(* IEC 61131-3 sources: Industry-PLC-LLM/data/PLCBEAD_repo/PLCBEAD_PLCEmbed-main/PLC-BEAD/Source/OpenPLCv2 (part 2) *)

(* ---- BAR_GRAPH.ST ---- *)
FUNCTION_BLOCK BAR_GRAPH
	VAR_INPUT
		X :	REAL;
		RST :	BOOL;
		TRIGGER_LOW :	REAL;
		TRIGGER_HIGH :	REAL;
		ALARM_LOW :	BOOL;
		ALARM_HIGH :	BOOL;
		LOG_SCALE :	BOOL;
	END_VAR

	VAR_OUTPUT
		LOW :	BOOL;
		Q1 :	BOOL;
		Q2 :	BOOL;
		Q3 :	BOOL;
		Q4 :	BOOL;
		Q5 :	BOOL;
		Q6 :	BOOL;
		HIGH :	BOOL;
		ALARM :	BOOL;
		STATUS :	BYTE;
	END_VAR

	VAR
		init :	BOOL;
		T1 :	REAL;
		T2 :	REAL;
		T3 :	REAL;
		T4 :	REAL;
		T5 :	REAL;
		temp :	REAL;
	END_VAR

	IF NOT init THEN
		init := TRUE;
		IF log_scale THEN
			temp := EXP(LN(Trigger_high / Trigger_low) * 0.166666666666666666666);
			T1 := trigger_low * temp;
			T2 := T1 * temp;
			T3 := T2 * temp;
			T4 := T3 * temp;
			T5 := T4 * temp;
		ELSE
			temp := (trigger_high - trigger_low) * 0.142857142;
			T1 := trigger_low + temp;
			T2 := T1 + temp;
			T3 := T2 + temp;
			T4 := T3 + temp;
			T5 := T4 + temp;
		END_IF;
	END_IF;

	Q1 := FALSE;
	Q2 := FALSE;
	Q3 := FALSE;
	Q4 := FALSE;
	Q5 := FALSE;
	Q6 := FALSE;
	status := BYTE#110;

	IF NOT alarm_low THEN low := FALSE; END_IF;
	IF NOT alarm_high THEN high := FALSE; END_IF;
	IF rst THEN
		alarm := FALSE;
		low := FALSE;
		high := FALSE;
	END_IF;

	IF X < trigger_low THEN
		Low := TRUE;
		status := BYTE#111;
		IF alarm_low THEN
			alarm := TRUE;
			status := BYTE#1;
		END_IF;
	ELSIF X < T1 THEN
		Q1 := TRUE;
	ELSIF x < t2 THEN
		Q2 := TRUE;
	ELSIF x < t3 THEN
		Q3 := TRUE;
	ELSIF x < T4 THEN
		Q4 := TRUE;
	ELSIF x < T5 THEN
		q5 := TRUE;
	ELSIF x < trigger_high THEN
		q6 := TRUE;
	ELSE
		high := TRUE;
		status := BYTE#112;
		IF alarm_high THEN
			alarm := TRUE;
			status := BYTE#2;
		END_IF;
	END_IF;

END_FUNCTION_BLOCK

PROGRAM program0
  VAR
    LocalVar0 : REAL;
    LocalVar1 : BOOL;
	LocalVar2 : REAL;
	LocalVar3 : REAL;
	LocalVar4 : BOOL;
	LocalVar5 : BOOL;
	LocalVar6 : BOOL;

	LOW   :	BOOL;
	Q1    :	BOOL;
	Q2    :	BOOL;
	Q3    :	BOOL;
	Q4    :	BOOL;
	Q5    :	BOOL;
	Q6    :	BOOL;
	HIGH  :	BOOL;
	ALARM :	BOOL;
	STATUS:	BYTE;

	func_block : BAR_GRAPH;
  END_VAR
	func_block.X := LocalVar0;
	func_block.RST := LocalVar1;
	func_block.TRIGGER_LOW := LocalVar2;
	func_block.TRIGGER_HIGH := LocalVar3;
	func_block.ALARM_LOW := LocalVar4;
	func_block.ALARM_HIGH := LocalVar5;
	func_block.LOG_SCALE := LocalVar6;

	func_block();
	LOW   := func_block.LOW   ;
	Q1    := func_block.Q1    ;
	Q2    := func_block.Q2    ;
	Q3    := func_block.Q3    ;
	Q4    := func_block.Q4    ;
	Q5    := func_block.Q5    ;
	Q6    := func_block.Q6    ;
	HIGH  := func_block.HIGH  ;
	ALARM := func_block.ALARM ;
	STATUS:= func_block.STATUS;

END_PROGRAM

CONFIGURATION Config0
  RESOURCE Res0 ON PLC
    TASK task0(INTERVAL := T#20ms,PRIORITY := 0);
    PROGRAM instance0 WITH task0 : program0;
  END_RESOURCE
END_CONFIGURATION

(* ---- BASE64_DECODE_STREAM.ST ---- *)
TYPE
  oscat_aB0_47	: ARRAY [0..47]	OF BYTE;
  oscat_aB0_63	: ARRAY [0..63]	OF BYTE;
END_TYPE

FUNCTION_BLOCK BASE64_DECODE_STREAM
	VAR_IN_OUT
		BUF1 :	oscat_aB0_63;
		BUF2 :	oscat_aB0_47;
	END_VAR

	VAR_INPUT
		SIZE1 :	INT;
	END_VAR

	VAR_OUTPUT
		SIZE2 :	INT;
	END_VAR

	VAR
		a :	INT;
		b :	WORD;
		o :	INT;
		off :	INT;
		i1 :	INT;
		i2 :	INT;
		c :	INT;
	END_VAR

	IF SIZE1 <= 0 THEN SIZE2 := 0; RETURN; END_IF;
	c := SIZE1 - 1;
	i2 := 0;
	a := 0;
	b := WORD#0;
	FOR i1 := 0 TO c DO
		o := BYTE_TO_INT(BUF1[i1]);
		IF o = 61  (* = *) THEN EXIT;
		ELSIF o > 96 (* a-z *) THEN off := 71;
		ELSIF o > 64 (* A-Z *) THEN off := 65;
		ELSIF o > 47 (* 0-9 *) THEN off := -4;
		ELSIF o = 43 (* + *) THEN off := -19;
		ELSIF o = 47 (* / *) THEN off := -16;
		END_IF;
		b := SHL(b,6) OR INT_TO_WORD(o - off);
		a := a + 6;
		IF a >= 8 THEN
			a := a - 8;
			BUF2[i2] := WORD_TO_BYTE(SHR(b,a));
			i2 := i2 + 1;
			b := b AND NOT SHL(WORD#16#FFFF,a);
		END_IF;
	END_FOR;
	SIZE2 := i2;
END_FUNCTION_BLOCK

PROGRAM program0
  VAR
	BUF1  :	oscat_aB0_63;
	BUF2  :	oscat_aB0_47;

	SIZE1 :	INT;

	SIZE2 :	INT;
	func_block : BASE64_DECODE_STREAM;
  END_VAR
	func_block.BUF1 :=BUF1 ;
	func_block.BUF2 :=BUF2 ;
	func_block.SIZE1:=SIZE1;
	func_block();
	BUF1 := func_block.BUF1;
	BUF2 := func_block.BUF2;
	SIZE2 := func_block.SIZE2;
END_PROGRAM

CONFIGURATION Config0
  RESOURCE Res0 ON PLC
    TASK task0(INTERVAL := T#20ms,PRIORITY := 0);
    PROGRAM instance0 WITH task0 : program0;
  END_RESOURCE
END_CONFIGURATION

(* ---- BLIND_ACTUATOR.ST ---- *)
FUNCTION_BLOCK INTERLOCK_Block

	VAR_INPUT
		I1 :	BOOL;
		I2 :	BOOL;
		TL :	TIME;
	END_VAR

	VAR_OUTPUT
		Q1 :	BOOL;
		Q2 :	BOOL;
	END_VAR

	VAR
		T1 :	TOF;
		T2 :	TOF;
	END_VAR

	T1(IN := I1, PT := TL);
	T2(IN := I2, PT := TL);

	Q1 := I1 AND NOT t2.Q;
	Q2 := I2 AND NOT t1.Q;

END_FUNCTION_BLOCK

FUNCTION TIME_TO_UDINT2:UDINT
	VAR_INPUT
		X :	TIME;
	END_VAR

	TIME_TO_UDINT2 := DINT_TO_UDINT(TIME_TO_DINT(X));
END_FUNCTION

FUNCTION_BLOCK T_PLC_MS_block
	VAR_OUTPUT
		T_PLC_MS :	UDINT;
	END_VAR

	VAR_EXTERNAL
		PLC_TICKS_PER_SEC :	INT;
		PLC_SYS_TICK_CNT :	DINT;
	END_VAR

	VAR
		debug :	BOOL;(*Debug-Mode ON / OFF*)
		N :	INT;(*Debug-Faktor*)
		Offset :	UDINT;(*Debug-Offset*)
		temp :	DWORD := DWORD#1;(*Debug-Offset*)
		mode :	BOOL;(*modus*)
		faktor :	UDINT;(*Systemtakt-Faktor*)
		init :	BOOL;
		v_plc_ticks_per_sec :	UDINT;
		base :	UDINT := UDINT#1000;
	END_VAR

	IF init = FALSE THEN
		v_plc_ticks_per_sec := INT_TO_UDINT(PLC_TICKS_PER_SEC);
		IF v_plc_ticks_per_sec = UDINT#1024 THEN
			faktor := UDINT#1;
			mode := FALSE;
		ELSIF v_plc_ticks_per_sec > UDINT#0 THEN
			IF v_plc_ticks_per_sec <= base THEN
				faktor := base / v_plc_ticks_per_sec;
				mode := FALSE;
			ELSE
				faktor := v_plc_ticks_per_sec / base;
				mode := TRUE;
			END_IF;
		ELSE
			faktor := UDINT#1;
		END_IF;
		init := TRUE;
	END_IF;

	IF mode THEN
		T_PLC_MS := DINT_TO_UDINT(PLC_SYS_TICK_CNT) / faktor;
	ELSE
		T_PLC_MS := DINT_TO_UDINT(PLC_SYS_TICK_CNT) * faktor;
	END_IF;

	IF debug THEN
		T_PLC_MS := (DWORD_TO_UDINT(SHL(UDINT_TO_DWORD(T_PLC_MS),N) OR SHL(temp,N)) - UDINT#1) + Offset;
	END_IF;
END_FUNCTION_BLOCK

FUNCTION FRMP_B:BYTE
	VAR_INPUT
		START :	BYTE;
		DIR :	BOOL;
		TD :	TIME;
		TR :	TIME;
	END_VAR

	IF TD < TR THEN
		FRMP_B := MIN(UDINT_TO_BYTE(DWORD_TO_UDINT(SHL(TIME_TO_DWORD(TD), 8)) / TIME_TO_UDINT2(TR)), SEL(DIR, START, USINT_TO_BYTE(USINT#255 - BYTE_TO_USINT(START))));
		IF DIR THEN
			FRMP_B := USINT_TO_BYTE(BYTE_TO_USINT(START) + BYTE_TO_USINT(FRMP_B));
		ELSE
			FRMP_B := USINT_TO_BYTE(BYTE_TO_USINT(START) - BYTE_TO_USINT(FRMP_B));
		END_IF;
	ELSE
		FRMP_B := SEL(DIR, BYTE#0, BYTE#255);
	END_IF;
END_FUNCTION

FUNCTION_BLOCK _RMP_B
	VAR_INPUT
		DIR :	BOOL;
		E :	BOOL := TRUE;
		TR :	TIME;
	END_VAR

	VAR_IN_OUT
		RMP :	BYTE;
	END_VAR

	VAR
		T_PLC_MS :	T_PLC_MS_block;
		tx :	TIME;
		tl :	TIME;
		tn :	TIME;
		init :	BOOL;
		last_dir :	BOOL;
		start :	BYTE;
	END_VAR

	T_PLC_MS();
	tx := UDINT_TO_TIME(T_PLC_MS.T_PLC_MS);

	IF E AND init AND (dir = last_dir) AND (RMP <> SEL(DIR, BYTE#0, BYTE#255)) AND TR = tn THEN
		RMP := FRMP_B(start, DIR, tx - tl, TR);
	ELSE
		init := TRUE;
		tl := tx;
		tn := tr;
		start := RMP;
	END_IF;
	last_dir := dir;
END_FUNCTION_BLOCK

FUNCTION_BLOCK RMP_B_Block

	VAR_INPUT
		SET :	BOOL;
		PT :	TIME;
		E :	BOOL := TRUE;
		UP :	BOOL := TRUE;
		RST :	BOOL;
	END_VAR

	VAR_OUTPUT
		OUT :	BYTE;
		BUSY :	BOOL;
		HIGH :	BOOL;
		LOW :	BOOL;
	END_VAR

	VAR
		rmp :	_RMP_B;
	END_VAR

	rmp(dir := UP, E := E, TR := PT, RMP := out);
	out := rmp.RMP;

	IF RST THEN
		out := BYTE#0;
	ELSIF SET THEN
		out := BYTE#255;
	END_IF;

low := out = BYTE#0;
high := out = BYTE#255;
busy := NOT (low OR high) AND E;

END_FUNCTION_BLOCK

FUNCTION_BLOCK BLIND_ACTUATOR_Block

	VAR_INPUT
		UP :	BOOL;
		DN :	BOOL;
		S_IN :	BYTE;
		T_UD :	TIME := T#10s;
		T_ANGLE :	TIME := T#3s;
		T_LOCKOUT :	TIME := t#100ms;
	END_VAR

	VAR_OUTPUT
		POS :	BYTE;
		ANG :	BYTE;
		QU :	BOOL;
		QD :	BOOL;
		STATUS :	BYTE;
	END_VAR

	VAR
		position :	RMP_B_Block;
		angle :	RMP_B_Block;
		lock :	INTERLOCK_Block;
	END_VAR

	lock(i1 := UP, I2 := DN, TL := T_lockout);

	angle(e := lock.Q1 OR lock.Q2, UP := lock.Q1, PT := T_Angle);
	position(e := lock.Q1 AND angle.high OR lock.Q2 AND angle.low, up := lock.Q1, PT := T_UD);

	pos := position.Out;
	ang := angle.Out;

	QU := lock.Q1;
	QD := lock.Q2;

	IF UP AND DN THEN
		status := BYTE#1;
	ELSIF UP THEN
		status := BYTE#121;
	ELSIF DN THEN
		status := BYTE#122;
	ELSE
		status := S_IN;
	END_IF;

END_FUNCTION_BLOCK

PROGRAM program0
	VAR
		UP :	BOOL;
		DN :	BOOL;
		S_IN :	BYTE;
		T_UD :	TIME := T#10s;
		T_ANGLE :	TIME := T#3s;
		T_LOCKOUT :	TIME := t#100ms;
		POS :	BYTE;
		ANG :	BYTE;
		QU :	BOOL;
		QD :	BOOL;
		func_block : BLIND_ACTUATOR_Block;
	END_VAR
	func_block.UP := UP;
	func_block.DN := DN;
	func_block.S_IN := S_IN ;
	func_block.T_UD := T_UD;
	func_block.T_ANGLE := T_ANGLE;
	func_block.T_LOCKOUT := T_LOCKOUT;
	func_block();
	POS  := func_block.POS;
	ANG  := func_block.ANG;
	QU  := func_block.QU;
	QD  := func_block.QD;
END_PROGRAM

CONFIGURATION Config0
	VAR_GLOBAL
		PLC_TICKS_PER_SEC :	INT;
		PLC_SYS_TICK_CNT :	DINT;
	END_VAR
  	RESOURCE Res0 ON PLC
    	TASK task0(INTERVAL := T#20ms,PRIORITY := 0);
    	PROGRAM instance0 WITH task0 : program0;
  	END_RESOURCE
END_CONFIGURATION

(* ---- BLIND_CONTROL.ST ---- *)
FUNCTION_BLOCK INTERLOCK_Block

	VAR_INPUT
		I1 :	BOOL;
		I2 :	BOOL;
		TL :	TIME;
	END_VAR

	VAR_OUTPUT
		Q1 :	BOOL;
		Q2 :	BOOL;
	END_VAR

	VAR
		T1 :	TOF;
		T2 :	TOF;
	END_VAR

	T1(IN := I1, PT := TL);
	T2(IN := I2, PT := TL);

	Q1 := I1 AND NOT t2.Q;
	Q2 := I2 AND NOT t1.Q;

END_FUNCTION_BLOCK

FUNCTION TIME_TO_UDINT2:UDINT
	VAR_INPUT
		X :	TIME;
	END_VAR

	TIME_TO_UDINT2 := DINT_TO_UDINT(TIME_TO_DINT(X));
END_FUNCTION

FUNCTION_BLOCK T_PLC_MS_block
	VAR_OUTPUT
		T_PLC_MS :	UDINT;
	END_VAR

	VAR_EXTERNAL
		PLC_TICKS_PER_SEC :	INT;
		PLC_SYS_TICK_CNT :	DINT;
	END_VAR

	VAR
		debug :	BOOL;(*Debug-Mode ON / OFF*)
		N :	INT;(*Debug-Faktor*)
		Offset :	UDINT;(*Debug-Offset*)
		temp :	DWORD := DWORD#1;(*Debug-Offset*)
		mode :	BOOL;(*modus*)
		faktor :	UDINT;(*Systemtakt-Faktor*)
		init :	BOOL;
		v_plc_ticks_per_sec :	UDINT;
		base :	UDINT := UDINT#1000;
	END_VAR

	IF init = FALSE THEN
		v_plc_ticks_per_sec := INT_TO_UDINT(PLC_TICKS_PER_SEC);
		IF v_plc_ticks_per_sec = UDINT#1024 THEN
			faktor := UDINT#1;
			mode := FALSE;
		ELSIF v_plc_ticks_per_sec > UDINT#0 THEN
			IF v_plc_ticks_per_sec <= base THEN
				faktor := base / v_plc_ticks_per_sec;
				mode := FALSE;
			ELSE
				faktor := v_plc_ticks_per_sec / base;
				mode := TRUE;
			END_IF;
		ELSE
			faktor := UDINT#1;
		END_IF;
		init := TRUE;
	END_IF;

	IF mode THEN
		T_PLC_MS := DINT_TO_UDINT(PLC_SYS_TICK_CNT) / faktor;
	ELSE
		T_PLC_MS := DINT_TO_UDINT(PLC_SYS_TICK_CNT) * faktor;
	END_IF;

	IF debug THEN
		T_PLC_MS := (DWORD_TO_UDINT(SHL(UDINT_TO_DWORD(T_PLC_MS),N) OR SHL(temp,N)) - UDINT#1) + Offset;
	END_IF;
END_FUNCTION_BLOCK

FUNCTION FRMP_B:BYTE
	VAR_INPUT
		START :	BYTE;
		DIR :	BOOL;
		TD :	TIME;
		TR :	TIME;
	END_VAR

	IF TD < TR THEN
		FRMP_B := MIN(UDINT_TO_BYTE(DWORD_TO_UDINT(SHL(TIME_TO_DWORD(TD), 8)) / TIME_TO_UDINT2(TR)), SEL(DIR, START, USINT_TO_BYTE(USINT#255 - BYTE_TO_USINT(START))));
		IF DIR THEN
			FRMP_B := USINT_TO_BYTE(BYTE_TO_USINT(START) + BYTE_TO_USINT(FRMP_B));
		ELSE
			FRMP_B := USINT_TO_BYTE(BYTE_TO_USINT(START) - BYTE_TO_USINT(FRMP_B));
		END_IF;
	ELSE
		FRMP_B := SEL(DIR, BYTE#0, BYTE#255);
	END_IF;
END_FUNCTION

FUNCTION_BLOCK _RMP_B
	VAR_INPUT
		DIR :	BOOL;
		E :	BOOL := TRUE;
		TR :	TIME;
	END_VAR

	VAR_IN_OUT
		RMP :	BYTE;
	END_VAR

	VAR
		T_PLC_MS :	T_PLC_MS_block;
		tx :	TIME;
		tl :	TIME;
		tn :	TIME;
		init :	BOOL;
		last_dir :	BOOL;
		start :	BYTE;
	END_VAR

	T_PLC_MS();
	tx := UDINT_TO_TIME(T_PLC_MS.T_PLC_MS);

	IF E AND init AND (dir = last_dir) AND (RMP <> SEL(DIR, BYTE#0, BYTE#255)) AND TR = tn THEN
		RMP := FRMP_B(start, DIR, tx - tl, TR);
	ELSE
		init := TRUE;
		tl := tx;
		tn := tr;
		start := RMP;
	END_IF;
	last_dir := dir;
END_FUNCTION_BLOCK

FUNCTION_BLOCK RMP_B_Block

	VAR_INPUT
		SET :	BOOL;
		PT :	TIME;
		E :	BOOL := TRUE;
		UP :	BOOL := TRUE;
		RST :	BOOL;
	END_VAR

	VAR_OUTPUT
		OUT :	BYTE;
		BUSY :	BOOL;
		HIGH :	BOOL;
		LOW :	BOOL;
	END_VAR

	VAR
		rmp :	_RMP_B;
	END_VAR

	rmp(dir := UP, E := E, TR := PT, RMP := out);
	out := rmp.RMP;

	IF RST THEN
		out := BYTE#0;
	ELSIF SET THEN
		out := BYTE#255;
	END_IF;

low := out = BYTE#0;
high := out = BYTE#255;
busy := NOT (low OR high) AND E;

END_FUNCTION_BLOCK

FUNCTION_BLOCK BLIND_ACTUATOR_Block

	VAR_INPUT
		UP :	BOOL;
		DN :	BOOL;
		S_IN :	BYTE;
		T_UD :	TIME := T#10s;
		T_ANGLE :	TIME := T#3s;
		T_LOCKOUT :	TIME := t#100ms;
	END_VAR

	VAR_OUTPUT
		POS :	BYTE;
		ANG :	BYTE;
		QU :	BOOL;
		QD :	BOOL;
		STATUS :	BYTE;
	END_VAR

	VAR
		position :	RMP_B_Block;
		angle :	RMP_B_Block;
		lock :	INTERLOCK_Block;
	END_VAR

	lock(i1 := UP, I2 := DN, TL := T_lockout);

	angle(e := lock.Q1 OR lock.Q2, UP := lock.Q1, PT := T_Angle);
	position(e := lock.Q1 AND angle.high OR lock.Q2 AND angle.low, up := lock.Q1, PT := T_UD);

	pos := position.Out;
	ang := angle.Out;

	QU := lock.Q1;
	QD := lock.Q2;

	IF UP AND DN THEN
		status := BYTE#1;
	ELSIF UP THEN
		status := BYTE#121;
	ELSIF DN THEN
		status := BYTE#122;
	ELSE
		status := S_IN;
	END_IF;

END_FUNCTION_BLOCK

FUNCTION _BYTE_TO_INT:INT
	VAR_INPUT
		IN :	BYTE;
	END_VAR

	_BYTE_TO_INT := USINT_TO_INT(BYTE_TO_USINT(IN));
END_FUNCTION

FUNCTION_BLOCK BLIND_CONTROL_Block

	VAR_INPUT
		UP :	BOOL;
		DN :	BOOL;
		S_IN :	BYTE;
		PI :	BYTE;
		AI :	BYTE;
		T_UD :	TIME;
		T_ANGLE :	TIME;
		SENS :	BYTE := 5;
		T_LOCKOUT :	TIME := T#100ms;
	END_VAR

	VAR_OUTPUT
		POS :	BYTE;
		ANG :	BYTE;
		MU :	BOOL;
		MD :	BOOL;
		STATUS :	BYTE;
	END_VAR

	VAR
		act :	BLIND_ACTUATOR_Block;
		delta :	BYTE;
		bTimeTest :	BOOL;
		iPos :	BYTE;
		iAngel :	BYTE;
	END_VAR

	IF bTimeTest THEN
		PI:=iPos;
		AI:=iAngel;
		UP:=TRUE;
		DN:=TRUE;
	END_IF;

	act(T_UD:=T_UD, T_ANGLE:=T_ANGLE, T_lockout := T_Lockout);

	IF UP AND DN THEN
		IF _BYTE_TO_INT(act.pos) < _BYTE_TO_INT(pi) - _BYTE_TO_INT(delta) THEN
			act.UP := TRUE;
			act.DN := FALSE;
			delta := BYTE#0;
			STATUS := BYTE#121;
		ELSIF _BYTE_TO_INT(act.pos) > _BYTE_TO_INT(pi) + _BYTE_TO_INT(delta) THEN
			act.UP := FALSE;
			act.DN := TRUE;
			delta := BYTE#0;
			STATUS := BYTE#122;
		ELSIF _BYTE_TO_INT(act.ang) < _BYTE_TO_INT(ai) - _BYTE_TO_INT(delta) AND T_angle > T#100ms THEN
			act.UP := TRUE;
			act.DN := FALSE;
			delta := SHR(sens,2);
			STATUS := BYTE#123;
		ELSIF _BYTE_TO_INT(act.ang) > _BYTE_TO_INT(ai) + _BYTE_TO_INT(delta) AND T_angle > T#100ms THEN
			act.UP := FALSE;
			act.DN := TRUE;
			delta := SHR(sens,2);
			STATUS := BYTE#124;
		ELSE
			act.UP := FALSE;
			act.DN := FALSE;
			delta := sens;
			STATUS := S_IN;
		END_IF;
	ELSE
		act.UP := UP;
		act.DN := DN;
		STATUS := S_IN;
	END_IF;

	act(T_UD:=T_UD, T_ANGLE:=T_ANGLE, T_lockout := T_Lockout);
	pos := act.pos;
	ang := act.ang;
	MU := act.QU;
	md := act.QD;
	status := act.status;

END_FUNCTION_BLOCK

PROGRAM program0
	VAR
		UP :	BOOL;
		DN :	BOOL;
		S_IN :	BYTE;
		PI :	BYTE;
		AI :	BYTE;
		T_UD :	TIME;
		T_ANGLE :	TIME;
		SENS :	BYTE := 5;
		T_LOCKOUT :	TIME := T#100ms;
		POS :	BYTE;
		ANG :	BYTE;
		MU :	BOOL;
		MD :	BOOL;
		STATUS :	BYTE;
		func_block : BLIND_CONTROL_Block;
	END_VAR
	func_block.UP := UP;
	func_block.DN := DN;
	func_block.S_IN := S_IN ;
	func_block.PI    := PI    ;
	func_block.AI := AI;
	func_block.T_UD := T_UD ;
	func_block.T_ANGLE    := T_ANGLE    ;
	func_block.SENS := SENS;
	func_block.T_LOCKOUT := T_LOCKOUT;
	func_block();
	POS  := func_block.POS;
	ANG  := func_block.ANG;
	MU  := func_block.MU;
	MD  := func_block.MD;
	STATUS  := func_block.STATUS;
END_PROGRAM

CONFIGURATION Config0
	VAR_GLOBAL
		PLC_TICKS_PER_SEC :	INT;
		PLC_SYS_TICK_CNT :	DINT;
	END_VAR
  	RESOURCE Res0 ON PLC
    	TASK task0(INTERVAL := T#20ms,PRIORITY := 0);
    	PROGRAM instance0 WITH task0 : program0;
  	END_RESOURCE
END_CONFIGURATION

(* ---- BLIND_CONTROL_S.ST ---- *)
FUNCTION UDINT_TO_TIME2:TIME

	VAR_INPUT
		IN :	UDINT;
	END_VAR

	UDINT_TO_TIME2 := DINT_TO_TIME(UDINT_TO_DINT(IN));

END_FUNCTION

FUNCTION_BLOCK T_PLC_MS_block
	VAR_OUTPUT
		T_PLC_MS :	UDINT;
	END_VAR

	VAR_EXTERNAL
		PLC_TICKS_PER_SEC :	INT;
		PLC_SYS_TICK_CNT :	DINT;
	END_VAR

	VAR
		debug :	BOOL;(*Debug-Mode ON / OFF*)
		N :	INT;(*Debug-Faktor*)
		Offset :	UDINT;(*Debug-Offset*)
		temp :	DWORD := DWORD#1;(*Debug-Offset*)
		mode :	BOOL;(*modus*)
		faktor :	UDINT;(*Systemtakt-Faktor*)
		init :	BOOL;
		v_plc_ticks_per_sec :	UDINT;
		base :	UDINT := UDINT#1000;
	END_VAR

	IF init = FALSE THEN
		v_plc_ticks_per_sec := INT_TO_UDINT(PLC_TICKS_PER_SEC);
		IF v_plc_ticks_per_sec = UDINT#1024 THEN
			faktor := UDINT#1;
			mode := FALSE;
		ELSIF v_plc_ticks_per_sec > UDINT#0 THEN
			IF v_plc_ticks_per_sec <= base THEN
				faktor := base / v_plc_ticks_per_sec;
				mode := FALSE;
			ELSE
				faktor := v_plc_ticks_per_sec / base;
				mode := TRUE;
			END_IF;
		ELSE
			faktor := UDINT#1;
		END_IF;
		init := TRUE;
	END_IF;

	IF mode THEN
		T_PLC_MS := DINT_TO_UDINT(PLC_SYS_TICK_CNT) / faktor;
	ELSE
		T_PLC_MS := DINT_TO_UDINT(PLC_SYS_TICK_CNT) * faktor;
	END_IF;

	IF debug THEN
		T_PLC_MS := (DWORD_TO_UDINT(SHL(UDINT_TO_DWORD(T_PLC_MS),N) OR SHL(temp,N)) - UDINT#1) + Offset;
	END_IF;
END_FUNCTION_BLOCK

FUNCTION TIME_TO_UDINT2:UDINT
	VAR_INPUT
		X :	TIME;
	END_VAR

	TIME_TO_UDINT2 := DINT_TO_UDINT(TIME_TO_DINT(X));
END_FUNCTION

FUNCTION FRMP_B:BYTE
	VAR_INPUT
		START :	BYTE;
		DIR :	BOOL;
		TD :	TIME;
		TR :	TIME;
	END_VAR

	IF TD < TR THEN
		FRMP_B := MIN(UDINT_TO_BYTE(DWORD_TO_UDINT(SHL(TIME_TO_DWORD(TD), 8)) / TIME_TO_UDINT2(TR)), SEL(DIR, START, USINT_TO_BYTE(USINT#255 - BYTE_TO_USINT(START))));
		IF DIR THEN
			FRMP_B := USINT_TO_BYTE(BYTE_TO_USINT(START) + BYTE_TO_USINT(FRMP_B));
		ELSE
			FRMP_B := USINT_TO_BYTE(BYTE_TO_USINT(START) - BYTE_TO_USINT(FRMP_B));
		END_IF;
	ELSE
		FRMP_B := SEL(DIR, BYTE#0, BYTE#255);
	END_IF;
END_FUNCTION

FUNCTION_BLOCK _RMP_B
	VAR_INPUT
		DIR :	BOOL;
		E :	BOOL := TRUE;
		TR :	TIME;
	END_VAR

	VAR_IN_OUT
		RMP :	BYTE;
	END_VAR

	VAR
		T_PLC_MS :	T_PLC_MS_block;
		tx :	TIME;
		tl :	TIME;
		tn :	TIME;
		init :	BOOL;
		last_dir :	BOOL;
		start :	BYTE;
	END_VAR

	T_PLC_MS();
	tx := UDINT_TO_TIME(T_PLC_MS.T_PLC_MS);

	IF E AND init AND (dir = last_dir) AND (RMP <> SEL(DIR, BYTE#0, BYTE#255)) AND TR = tn THEN
		RMP := FRMP_B(start, DIR, tx - tl, TR);
	ELSE
		init := TRUE;
		tl := tx;
		tn := tr;
		start := RMP;
	END_IF;
	last_dir := dir;
END_FUNCTION_BLOCK

FUNCTION_BLOCK TREND_DW
	VAR_INPUT
		X :	DWORD;
	END_VAR
	VAR_OUTPUT
		Q :	BOOL;
		TU :	BOOL;
		TD :	BOOL;
		D :	DWORD;
	END_VAR

	VAR
		LAST_X :	DWORD;
	END_VAR

	IF X > last_X THEN
		TU := TRUE;
		TD := FALSE;
		D := UDINT_TO_DWORD(DWORD_TO_UDINT(X) - DWORD_TO_UDINT(last_X));
		Q := TRUE;
	ELSIF X < last_X THEN
		TD := TRUE;
		TU := FALSE;
		D := UDINT_TO_DWORD(DWORD_TO_UDINT(last_X) - DWORD_TO_UDINT(X));
		Q := FALSE;
	ELSE
		TU := FALSE;
		TD := FALSE;
		D := DWORD#0;
	END_IF;
	last_X := X;
END_FUNCTION_BLOCK

FUNCTION_BLOCK _RMP_NEXT
	VAR_INPUT
		E :	BOOL := TRUE;
		IN :	BYTE;
		TR :	TIME;
		TF :	TIME;
		TL :	TIME;
	END_VAR

	VAR_OUTPUT
		DIR :	BOOL;
		UP :	BOOL;
		DN :	BOOL;
	END_VAR

	VAR_IN_OUT
		OUT :	BYTE;
	END_VAR
	VAR
		rmx :	_RMP_B;
		dirx :	TREND_DW;
		t_lock :	TP;
		xen :	BOOL;
		xdir :	BOOL;
	END_VAR

	dirx(X := BYTE_TO_DWORD(in));

	t_lock(in := FALSE, pt := TL);

	IF dirx.TU AND (OUT < IN) THEN
		IF NOT xdir AND xen THEN t_lock(in := TRUE); END_IF;
		xen := TRUE;
		xdir := TRUE;
	ELSIF dirx.TD AND (OUT > IN) THEN
		IF xdir AND xen THEN t_lock(in := TRUE); END_IF;
		xen := TRUE;
		xdir := FALSE;
	ELSIF xen THEN
		IF (xdir AND (out >= in)) OR (NOT xdir AND (out <= in)) THEN
			xen := FALSE;
			IF tl > t#0s THEN t_lock(IN := TRUE); END_IF;
		END_IF;
	END_IF;

	IF NOT t_lock.Q AND xen THEN
		UP := XDIR;
		DIR := XDIR;
		DN := NOT XDIR;
	ELSE
		UP := FALSE;
		DN := FALSE;
	END_IF;

	rmx(rmp := OUT, E := E AND (UP OR DN) , dir := DIR, tr := SEL(dir, TF, TR));
	OUT := rmx.RMP;
END_FUNCTION_BLOCK

FUNCTION _BYTE_TO_INT:INT
	VAR_INPUT
		IN :	BYTE;
	END_VAR

	_BYTE_TO_INT := USINT_TO_INT(BYTE_TO_USINT(IN));
END_FUNCTION

FUNCTION_BLOCK BLIND_CONTROL_S_Block

	VAR_INPUT
		UP :	BOOL;
		DN :	BOOL;
		S_IN :	BYTE := BYTE#125;
		PI :	BYTE;
		T_UP :	TIME;
		T_DN :	TIME;
		RU :	BOOL;
		RD :	BOOL;
		T_LOCKOUT :	TIME := T#100ms;
		T_EXT :	TIME;
		EXT_TRIG :	BYTE := BYTE#5;
		R_POS_TOP :	BYTE := BYTE#255;
		R_POS_BOT :	BYTE;
	END_VAR

	VAR_OUTPUT
		POS :	BYTE;
		MU :	BOOL;
		MD :	BOOL;
		STATUS :	BYTE;
	END_VAR

	VAR
		T_PLC_MS :	T_PLC_MS_Block;
		rmp :	_RMP_NEXT;
		tx :	TIME;
		last :	TIME;
		pi_last :	BYTE;
	END_VAR

	T_PLC_MS();
	tx:= UDINT_TO_TIME(T_PLC_MS.T_PLC_MS);

	IF UP  AND NOT DN THEN
		rmp.IN := BYTE#255;
		STATUS := BYTE#121;
	ELSIF DN AND NOT UP THEN
		rmp.IN := BYTE#0;
		STATUS := BYTE#122;
	ELSIF NOT (UP OR DN) THEN
		rmp.IN := PI;
		STATUS := S_IN;
	END_IF;

	rmp(E := UP OR DN, TR := T_UP, TF := T_DN, TL := T_LOCKOUT, OUT := POS);
	pos := rmp.OUT;

	CASE _BYTE_TO_INT(STATUS) OF
		0:
			last := tx;
			PI_last := PI XOR BYTE#255;
			STATUS := BYTE#128;

		121:
			MU := TRUE;
			MD := FALSE;
			IF POS >= USINT_TO_BYTE(USINT#255 - BYTE_TO_USINT(EXT_TRIG)) THEN
				POS := BYTE#255;
				last := tx;
				STATUS := BYTE#129;
			END_IF;

		122:
			MD := TRUE;
			MU := FALSE;
			IF POS <= EXT_TRIG THEN
				POS := BYTE#0;
				last := tx;
				STATUS := BYTE#129;
			END_IF;

		123:
			MD := rmp.DN;
			MU := rmp.UP;
			IF NOT (rmp.DN OR rmp.UP) THEN
				IF POS <= EXT_TRIG THEN
					MD := TRUE;
					last := tx;
					STATUS := BYTE#129;
				ELSIF POS >= USINT_TO_BYTE(USINT#255 - BYTE_TO_USINT(EXT_TRIG)) THEN
					MU := TRUE;
					last := tx;
					STATUS := BYTE#129;
				ELSE
					STATUS := S_IN;
				END_IF;
			END_IF;

		124:
			MD := rmp.DN;
			MU := rmp.UP;
			IF NOT(rmp.DN OR rmp.UP) THEN
				PI_last := PI;
				STATUS := S_IN;
			END_IF;

		127:
			IF (tx - last) >= T_LOCKOUT THEN
					STATUS := S_IN;
			END_IF;

		128:
			MU := TRUE;
			MD := FALSE;
			rmp.IN := BYTE#255;
			IF (tx - last) >= (T_UP +  T_EXT) THEN
				MU := FALSE;
				last := tx;
				STATUS := BYTE#127;
			END_IF;

		129:
			IF (tx - last) >= T_EXT THEN
				MU := FALSE;
				MD := FALSE;
				last := tx;
				STATUS := BYTE#127;
			END_IF;

	ELSE
		MU := FALSE;
		MD := FALSE;
		IF PI <> PI_last THEN
			PI_last := PI;
			rmp.IN := PI;
			STATUS := BYTE#123;
		ELSIF POS = BYTE#0 AND RU THEN
			rmp.IN := R_POS_BOT;
			STATUS := BYTE#124;
		ELSIF pos = BYTE#255 AND RD THEN
			rmp.IN := R_POS_TOP;
			STATUS := BYTE#124;
		ELSE
			STATUS := S_IN;
		END_IF;
	END_CASE;

END_FUNCTION_BLOCK

PROGRAM program0
	VAR
		UP :	BOOL;
		DN :	BOOL;
		S_IN :	BYTE := BYTE#125;
		PI :	BYTE;
		T_UP :	TIME;
		T_DN :	TIME;
		RU :	BOOL;
		RD :	BOOL;
		T_LOCKOUT :	TIME := T#100ms;
		T_EXT :	TIME;
		EXT_TRIG :	BYTE := BYTE#5;
		R_POS_TOP :	BYTE := BYTE#255;
		R_POS_BOT :	BYTE;
		POS :	BYTE;
		MU :	BOOL;
		MD :	BOOL;
		STATUS :	BYTE;
		func_block : BLIND_CONTROL_S_Block;
	END_VAR
	func_block.UP := UP;
	func_block.DN := DN;
	func_block.S_IN := S_IN ;
	func_block.PI    := PI    ;
	func_block.T_UP := T_UP;
	func_block.T_DN := T_DN ;
	func_block.RU    := RU    ;
	func_block.RD := RD;
	func_block.T_LOCKOUT := T_LOCKOUT;
	func_block.T_EXT := T_EXT ;
	func_block.EXT_TRIG    := EXT_TRIG    ;
	func_block.R_POS_TOP := R_POS_TOP;
	func_block.R_POS_BOT := R_POS_BOT ;
	func_block();
	POS  := func_block.POS;
	MU  := func_block.MU;
	MD  := func_block.MD;
	STATUS  := func_block.STATUS;
END_PROGRAM

CONFIGURATION Config0
	VAR_GLOBAL
		PLC_TICKS_PER_SEC :	INT;
		PLC_SYS_TICK_CNT :	DINT;
	END_VAR
  	RESOURCE Res0 ON PLC
    	TASK task0(INTERVAL := T#20ms,PRIORITY := 0);
    	PROGRAM instance0 WITH task0 : program0;
  	END_RESOURCE
END_CONFIGURATION

(* ---- BLIND_INPUT.ST ---- *)
FUNCTION UDINT_TO_TIME2:TIME

	VAR_INPUT
		IN :	UDINT;
	END_VAR

	UDINT_TO_TIME2 := DINT_TO_TIME(UDINT_TO_DINT(IN));

END_FUNCTION

FUNCTION_BLOCK T_PLC_MS_block
	VAR_OUTPUT
		T_PLC_MS :	UDINT;
	END_VAR

	VAR_EXTERNAL
		PLC_TICKS_PER_SEC :	INT;
		PLC_SYS_TICK_CNT :	DINT;
	END_VAR

	VAR
		debug :	BOOL;(*Debug-Mode ON / OFF*)
		N :	INT;(*Debug-Faktor*)
		Offset :	UDINT;(*Debug-Offset*)
		temp :	DWORD := DWORD#1;(*Debug-Offset*)
		mode :	BOOL;(*modus*)
		faktor :	UDINT;(*Systemtakt-Faktor*)
		init :	BOOL;
		v_plc_ticks_per_sec :	UDINT;
		base :	UDINT := UDINT#1000;
	END_VAR

	IF init = FALSE THEN
		v_plc_ticks_per_sec := INT_TO_UDINT(PLC_TICKS_PER_SEC);
		IF v_plc_ticks_per_sec = UDINT#1024 THEN
			faktor := UDINT#1;
			mode := FALSE;
		ELSIF v_plc_ticks_per_sec > UDINT#0 THEN
			IF v_plc_ticks_per_sec <= base THEN
				faktor := base / v_plc_ticks_per_sec;
				mode := FALSE;
			ELSE
				faktor := v_plc_ticks_per_sec / base;
				mode := TRUE;
			END_IF;
		ELSE
			faktor := UDINT#1;
		END_IF;
		init := TRUE;
	END_IF;

	IF mode THEN
		T_PLC_MS := DINT_TO_UDINT(PLC_SYS_TICK_CNT) / faktor;
	ELSE
		T_PLC_MS := DINT_TO_UDINT(PLC_SYS_TICK_CNT) * faktor;
	END_IF;

	IF debug THEN
		T_PLC_MS := (DWORD_TO_UDINT(SHL(UDINT_TO_DWORD(T_PLC_MS),N) OR SHL(temp,N)) - UDINT#1) + Offset;
	END_IF;

END_FUNCTION_BLOCK

FUNCTION_BLOCK CLICK_MODE_Block

	VAR_INPUT
		IN :	BOOL;
		T_LONG :	TIME := T#500ms;
	END_VAR

	VAR_OUTPUT
		SINGLE :	BOOL;
		DOUBLE :	BOOL;
		LONG :	BOOL;
		TP_LONG :	BOOL;
	END_VAR

	VAR
		Timer :	TP;
		cnt :	INT;
		last :	BOOL;
	END_VAR

	timer(in := IN, PT := T_LONG);
	single := FALSE;
	double := FALSE;

	IF timer.Q THEN
		IF NOT in AND last THEN	cnt := cnt + 1; END_IF;
	ELSE
		CASE cnt OF
			1 : single := TRUE;
			2 : double := TRUE;
		END_CASE;
		cnt := 0;
	END_IF;
	last := in;
	TP_LONG := NOT timer.Q AND (NOT LONG) AND IN;
	LONG := NOT timer.Q AND in;

END_FUNCTION_BLOCK

FUNCTION _BYTE_TO_INT:INT
	VAR_INPUT
		IN :	BYTE;
	END_VAR

	_BYTE_TO_INT := USINT_TO_INT(BYTE_TO_USINT(IN));
END_FUNCTION

FUNCTION_BLOCK BLIND_INPUT_Block

	VAR_INPUT
		POS :	BYTE;
		ANG :	BYTE;
		S1 :	BOOL;
		S2 :	BOOL;
		IN :	BOOL;
		PI :	BYTE;
		AI :	BYTE;
		SINGLE_SWITCH :	BOOL;
		CLICK_EN :	BOOL := TRUE;
		CLICK_TIME :	TIME := T#500ms;
		MAX_RUNTIME :	TIME := T#60s;
		MANUAL_TIMEOUT :	TIME := T#1h;
		DEBOUNCE_TIME :	TIME := T#20ms;
		DBL_CLK1 :	BOOL := FALSE;
		DBL_POS1 :	BYTE;
		DBL_ANG1 :	BYTE;
		DBL_CLK2 :	BOOL := FALSE;
		DBL_POS2 :	BYTE := BYTE#255;
		DBL_ANG2 :	BYTE := BYTE#255;
		D1_TOGGLE :	BOOL := TRUE;
		D2_TOGGLE :	BOOL := TRUE;
		MASTER_MODE :	BOOL;
	END_VAR

	VAR_OUTPUT
		QU :	BOOL := TRUE;
		QD :	BOOL := TRUE;
		STATUS :	BYTE;
		PO :	BYTE := BYTE#255;
		AO :	BYTE := BYTE#255;
		D1 :	BOOL;
		D2 :	BOOL;
	END_VAR

	VAR
		s1e :	TOF;
		s2e :	TOF;
		s1d :	CLICK_MODE_Block;
		s2d :	CLICK_MODE_Block;
		dir :	BOOL;
		tx :	TIME;
		last :	TIME;
		T_PLC_MS :	T_PLC_MS_Block;
	END_VAR

	T_PLC_MS();
	tx:= UDINT_TO_TIME(T_PLC_MS.T_PLC_MS);

	s1e(in := S1, pt := DEBOUNCE_TIME);
	s2e(in := S2, pt := DEBOUNCE_TIME);
	s1d(in := (s1e.Q AND NOT SINGLE_SWITCH) OR (s1e.Q AND SINGLE_SWITCH AND dir), t_long := CLICK_TIME);
	s2d(in := (s2e.Q AND NOT SINGLE_SWITCH) OR (s1e.Q AND SINGLE_SWITCH AND NOT dir), t_long := CLICK_TIME);

	IF NOT d1_toggle THEN d1 := FALSE; END_IF;
	IF NOT d2_toggle THEN d2 := FALSE; END_IF;

	IF (s1d.LONG AND s2d.LONG) OR (status = BYTE#139) THEN
	status := BYTE#139;
	IF NOT (s1d.LONG OR s2d.LONG)  THEN status := BYTE#130; END_IF;
	ELSIF s1d.tp_LONG THEN
		status := BYTE#132;
	ELSIF s2d.tp_LONG THEN
		status := BYTE#133;
	ELSIF  s1d.SINGLE THEN
		IF click_en THEN
			IF QU XOR QD THEN
				status := BYTE#131;
			ELSE
				status := BYTE#134;
				last := tx;
				dir := NOT dir;
			END_IF;
		END_IF;
	ELSIF  s2d.SINGLE THEN
		IF click_en THEN
			IF QU XOR QD THEN
				status := BYTE#131;
			ELSE
				status := BYTE#135;
				last := tx;
				dir := NOT dir;
			END_IF;
		END_IF;
	ELSIF in THEN
		status := BYTE#136;
		last := tx;
	ELSIF s1d.DOUBLE THEN
		IF dbl_clk1 THEN
			status := BYTE#137;
			last := tx;
		ELSE
			D1 := NOT D1;
		END_IF;
	ELSIF s2d.DOUBLE THEN
		IF dbl_clk2 THEN
			status := BYTE#138;
			last := tx;
		ELSE
			IF single_switch THEN D1 := NOT D1; ELSE D2 := NOT D2; END_IF;
		END_IF;
	END_IF;

	CASE _BYTE_TO_INT(status) OF
		0:
				status := BYTE#130;

		130:
				IF NOT master_mode THEN
					PO := POS;
					AO := ANG;
				END_IF;
				QU := TRUE;
				QD := TRUE;

		131:
				QU := FALSE;
				QD := FALSE;
				PO := POS;
				AO := ANG;
				IF tx - last >= manual_timeout THEN
					status := BYTE#130;
				END_IF;

		132:
				QU := TRUE;
				QD := FALSE;
				PO := POS; AO := ANG;
				last := tx;
				IF NOT s1d.LONG THEN status := BYTE#131; dir := NOT dir; END_IF;

		133:
				QU := FALSE;
				QD := TRUE;
				PO := POS; AO := ANG;
				last := tx;
				IF NOT s2d.LONG THEN	status := BYTE#131; dir := NOT dir; END_IF;

		134:
				QU := TRUE;
				QD := FALSE;
				PO := POS; AO := ANG;
				IF tx - last >= max_runtime THEN status := BYTE#131; END_IF;

		135:
				QU := FALSE;
				QD := TRUE;
				PO := POS; AO := ANG;
				IF tx - last >= max_runtime THEN status := BYTE#131;	END_IF;

		136:
				QU := TRUE;
				QD := TRUE;
				PO := PI; AO := AI;
				IF tx-last >= max_runtime THEN status := BYTE#130; END_IF;

		137:
				QU := TRUE;
				QD := TRUE;
				PO := DBL_POS1;
				AO := DBL_ANG1;
				IF tx - last >= max_runtime THEN status := BYTE#131; END_IF;

		138:
				QU := TRUE;
				QD := TRUE;
				PO := DBL_POS2;
				AO := DBL_ANG2;
				IF tx - last >= max_runtime THEN status := BYTE#131; END_IF;

		139:
				QU := FALSE;
				QD := FALSE;
				PO := POS;
				AO := ANG;

	END_CASE;

END_FUNCTION_BLOCK

PROGRAM program0
	VAR
		POS :	BYTE;
		ANG :	BYTE;
		S1 :	BOOL;
		S2 :	BOOL;
		IN :	BOOL;
		PI :	BYTE;
		AI :	BYTE;
		SINGLE_SWITCH :	BOOL;
		CLICK_EN :	BOOL := TRUE;
		CLICK_TIME :	TIME := T#500ms;
		MAX_RUNTIME :	TIME := T#60s;
		MANUAL_TIMEOUT :	TIME := T#1h;
		DEBOUNCE_TIME :	TIME := T#20ms;
		DBL_CLK1 :	BOOL := FALSE;
		DBL_POS1 :	BYTE;
		DBL_ANG1 :	BYTE;
		DBL_CLK2 :	BOOL := FALSE;
		DBL_POS2 :	BYTE := BYTE#255;
		DBL_ANG2 :	BYTE := BYTE#255;
		D1_TOGGLE :	BOOL := TRUE;
		D2_TOGGLE :	BOOL := TRUE;
		MASTER_MODE :	BOOL;
		QU :	BOOL := TRUE;
		QD :	BOOL := TRUE;
		STATUS :	BYTE;
		PO :	BYTE := BYTE#255;
		AO :	BYTE := BYTE#255;
		D1 :	BOOL;
		D2 :	BOOL;
		func_block : BLIND_INPUT_Block;
	END_VAR
	func_block.POS := POS;
	func_block.ANG := ANG;
	func_block.S1 := S1 ;
	func_block.S2 := S2;
	func_block.IN := IN;
	func_block.PI := PI;
	func_block.AI := AI;
	func_block.SINGLE_SWITCH := SINGLE_SWITCH;
	func_block.CLICK_EN := CLICK_EN ;
	func_block.CLICK_TIME := CLICK_TIME;
	func_block.MAX_RUNTIME := MAX_RUNTIME;
	func_block.MANUAL_TIMEOUT := MANUAL_TIMEOUT;
	func_block.DEBOUNCE_TIME := DEBOUNCE_TIME;
	func_block.DBL_CLK1 := DBL_CLK1;
	func_block.DBL_POS1 := DBL_POS1 ;
	func_block.DBL_ANG1 := DBL_ANG1;
	func_block.DBL_CLK2 := DBL_CLK2;
	func_block.DBL_POS2 := DBL_POS2;
	func_block.DBL_ANG2 := DBL_ANG2;
	func_block.D1_TOGGLE := D1_TOGGLE ;
	func_block.D2_TOGGLE := D2_TOGGLE;
	func_block.MASTER_MODE := MASTER_MODE;
	func_block();
	QU  := func_block.QU;
	QD  := func_block.QD;
	STATUS  := func_block.STATUS;
	PO  := func_block.PO;
	AO  := func_block.AO;
	D1  := func_block.D1;
	D2  := func_block.D2;
END_PROGRAM

CONFIGURATION Config0
	VAR_GLOBAL
		PLC_TICKS_PER_SEC :	INT;
		PLC_SYS_TICK_CNT :	DINT;
	END_VAR
  	RESOURCE Res0 ON PLC
    	TASK task0(INTERVAL := T#20ms,PRIORITY := 0);
    	PROGRAM instance0 WITH task0 : program0;
  	END_RESOURCE
END_CONFIGURATION

(* ---- BLIND_NIGHT.ST ---- *)
FUNCTION TIME_TO_UDINT2:UDINT
	VAR_INPUT
		X :	TIME;
	END_VAR

	TIME_TO_UDINT2 := DINT_TO_UDINT(TIME_TO_DINT(X));
END_FUNCTION

FUNCTION DT_TO_DATE2:UDINT

	VAR_INPUT
		IN :	UDINT;
	END_VAR

	DT_TO_DATE2 := (IN / UDINT#86400) * UDINT#86400;
END_FUNCTION

FUNCTION DT_TO_TOD2:UDINT
	VAR_INPUT
		IN :	UDINT;
	END_VAR

	DT_TO_TOD2 := (IN MOD UDINT#86400) * UDINT#1000;
END_FUNCTION

FUNCTION_BLOCK BLIND_NIGHT_Block

	VAR_INPUT
		UP :	BOOL;
		DN :	BOOL;
		S_IN :	BYTE;
		PI :	BYTE;
		AI :	BYTE;
		E_NIGHT :	BOOL := TRUE;
		E_DAY :	BOOL := TRUE;
		DTIN :	UDINT;
		SUNRISE :	UDINT;
		SUNSET :	UDINT;
		SUNRISE_OFFSET :	TIME;
		SUNSET_OFFSET :	TIME;
		NIGHT_POSITION :	BYTE;
		NIGHT_ANGLE :	BYTE;
	END_VAR

	VAR_OUTPUT
		QU :	BOOL;
		QD :	BOOL;
		STATUS :	BYTE;
		PO :	BYTE;
		AO :	BYTE;
	END_VAR

	VAR
		night :	BOOL;
		last_night :	UDINT;
		last_day :	UDINT;
	END_VAR

	IF NOT (up AND dn) AND night THEN
		night := FALSE;
	ELSIF (DT_TO_TOD2(dtin) > sunset + TIME_TO_UDINT2(sunset_offset)) AND (last_night < DT_TO_DATE2(dtin)) AND NOT night AND e_night THEN
		night := TRUE;
		last_night := DT_TO_DATE2(dtin);
	ELSIF (DT_TO_TOD2(dtin) > sunrise + TIME_TO_UDINT2(sunrise_offset)) AND (last_day < DT_TO_DATE2(dtin)) AND night AND e_day AND (last_night < DT_TO_DATE2(dtin)) THEN
		night := FALSE;
		last_day := DT_TO_DATE2(dtin);
	END_IF;

	IF UP AND DN AND night THEN
		status := BYTE#141;
		po := night_position;
		ao := night_angle;
	ELSE
		QU := UP;
		QD := DN;
		po := pi;
		ao := ai;
		status := s_in;
	END_IF;

END_FUNCTION_BLOCK

PROGRAM program0
	VAR
		UP :	BOOL;
		DN :	BOOL;
		S_IN :	BYTE;
		PI :	BYTE;
		AI :	BYTE;
		E_NIGHT :	BOOL := TRUE;
		E_DAY :	BOOL := TRUE;
		DTIN :	UDINT;
		SUNRISE :	UDINT;
		SUNSET :	UDINT;
		SUNRISE_OFFSET :	TIME;
		SUNSET_OFFSET :	TIME;
		NIGHT_POSITION :	BYTE;
		NIGHT_ANGLE :	BYTE;
		QU :	BOOL;
		QD :	BOOL;
		STATUS :	BYTE;
		PO :	BYTE;
		AO :	BYTE;

		func_block : BLIND_NIGHT_Block;
	END_VAR
	func_block.UP := UP;
	func_block.DN := DN;
	func_block.S_IN := S_IN ;
	func_block.PI    := PI    ;
	func_block.AI := AI;
	func_block.E_NIGHT := E_NIGHT;
	func_block.E_DAY := E_DAY ;
	func_block.DTIN    := DTIN    ;
	func_block.SUNRISE := SUNRISE;
	func_block.SUNSET := SUNSET;
	func_block.SUNRISE_OFFSET := SUNRISE_OFFSET ;
	func_block.SUNSET_OFFSET    := SUNSET_OFFSET    ;
	func_block.NIGHT_POSITION := NIGHT_POSITION ;
	func_block.NIGHT_ANGLE    := NIGHT_ANGLE    ;

	func_block();
	QU  := func_block.QU;
	QD  := func_block.QD;
	STATUS  := func_block.STATUS;
	PO  := func_block.PO;
	AO  := func_block.AO;
END_PROGRAM

CONFIGURATION Config0
	RESOURCE Res0 ON PLC
		TASK task0(INTERVAL := T#20ms,PRIORITY := 0);
		PROGRAM instance0 WITH task0 : program0;
	END_RESOURCE
END_CONFIGURATION

(* ---- BLIND_SCENE.ST ---- *)
TYPE
	oscat_bsa_X                 : ARRAY [0..2]    OF BYTE;
  	oscat_blind_scene_array     : ARRAY [0..15]   OF oscat_bsa_X := [0, 0, 0, 0, 0, 0, 0, 0, 0, 0, 0, 0, 0, 0, 0, 0];
END_TYPE

FUNCTION _BYTE_TO_INT:INT
	VAR_INPUT
		IN :	BYTE;
	END_VAR

	_BYTE_TO_INT := USINT_TO_INT(BYTE_TO_USINT(IN));
END_FUNCTION

FUNCTION_BLOCK BLIND_SCENE_Block

	VAR_INPUT
		UP :	BOOL;
		DN :	BOOL;
		S_IN :	BYTE;
		PI :	BYTE;
		AI :	BYTE;
		ENABLE :	BOOL;
		SWRITE :	BOOL;
		SCENE :	BYTE;
	END_VAR

	VAR_OUTPUT
		QU :	BOOL;
		QD :	BOOL;
		STATUS :	BYTE;
		PO :	BYTE;
		AO :	BYTE;
	END_VAR

	VAR
		x :	INT;
	END_VAR

	VAR RETAIN
		sx :	oscat_blind_scene_array;
	END_VAR

	x := _BYTE_TO_INT(scene AND BYTE#2#0000_1111);

	IF enable AND (sx[x][2] > BYTE#0) AND UP AND DN THEN
		po := sx[x][0];
		ao := sx[x][1];
		status := INT_TO_BYTE(160 + x);
		QU := TRUE;
		QD := TRUE;
	ELSE
		QU := UP;
		QD := DN;
		status := S_IN;
		po := pi;
		ao := ai;
	END_IF;

	IF swrite THEN
		status := BYTE#176;
		sx[x][0] := pi;
		sx[x][1] := ai;
		IF enable THEN sx[x][2] := BYTE#1; ELSE sx[x][2] := BYTE#0; END_IF;
	END_IF;

END_FUNCTION_BLOCK

PROGRAM program0
	VAR
		UP :	BOOL;
		DN :	BOOL;
		S_IN :	BYTE;
		PI :	BYTE;
		AI :	BYTE;
		ENABLE :	BOOL;
		SWRITE :	BOOL;
		SCENE :	BYTE;
		QU :	BOOL;
		QD :	BOOL;
		STATUS :	BYTE;
		PO :	BYTE;
		AO :	BYTE;

		func_block : BLIND_SCENE_Block;
	END_VAR
	func_block.UP := UP;
	func_block.DN := DN;
	func_block.S_IN := S_IN ;
	func_block.PI    := PI    ;
	func_block.AI := AI;
	func_block.ENABLE := ENABLE;
	func_block.SWRITE := SWRITE ;
	func_block.SCENE := SCENE ;

	func_block();
	QU  := func_block.QU;
	QD  := func_block.QD;
	STATUS  := func_block.STATUS;
	PO  := func_block.PO;
	AO  := func_block.AO;
END_PROGRAM

CONFIGURATION Config0
	RESOURCE Res0 ON PLC
		TASK task0(INTERVAL := T#20ms,PRIORITY := 0);
		PROGRAM instance0 WITH task0 : program0;
	END_RESOURCE
END_CONFIGURATION

(* ---- BLIND_SECURITY.ST ---- *)
FUNCTION_BLOCK BLIND_SECURITY_Block

	VAR_INPUT
		UP :	BOOL;
		DN :	BOOL;
		S_IN :	BYTE;
		PI :	BYTE;
		AI :	BYTE;
		FIRE :	BOOL;
		WIND :	BOOL;
		ALARM :	BOOL;
		DOOR :	BOOL;
		RAIN :	BOOL;
		ALARM_UP :	BOOL := TRUE;
		WIND_UP :	BOOL := TRUE;
		RAIN_UP :	BOOL := TRUE;
	END_VAR

	VAR_OUTPUT
		QU :	BOOL;
		QD :	BOOL;
		STATUS :	BYTE;
		PO :	BYTE;
		AO :	BYTE;
	END_VAR

	IF Fire THEN
		QU := TRUE;
		QD := FALSE;
		status := BYTE#111;
	ELSIF Wind THEN
		QU := Wind_up;
		QD := NOT wind_up;
		status := BYTE#112;
	ELSIF alarm THEN
		QU := Alarm_up;
		QD := NOT Alarm_up;
		status := BYTE#113;
	ELSIF Door THEN
		QU := TRUE;
		QD := FALSE;
		status := BYTE#114;
	ELSIF Rain AND NOT (up XOR dn) THEN
		QU := rain_up;
		QD := NOT rain_up;
		status := BYTE#115;
	ELSE
		QU := UP;
		QD := DN;
		status := S_IN;
		po := pi;
		ao := ai;
	END_IF;

END_FUNCTION_BLOCK

PROGRAM program0
	VAR
		UP :	BOOL;
		DN :	BOOL;
		S_IN :	BYTE;
		PI :	BYTE;
		AI :	BYTE;
		FIRE :	BOOL;
		WIND :	BOOL;
		ALARM :	BOOL;
		DOOR :	BOOL;
		RAIN :	BOOL;
		ALARM_UP :	BOOL := TRUE;
		WIND_UP :	BOOL := TRUE;
		RAIN_UP :	BOOL := TRUE;
		QU :	BOOL;
		QD :	BOOL;
		STATUS :	BYTE;
		PO :	BYTE;
		AO :	BYTE;

		func_block : BLIND_SECURITY_Block;
	END_VAR
	func_block.UP := UP;
	func_block.DN := DN;
	func_block.S_IN := S_IN ;
	func_block.PI    := PI    ;
	func_block.AI := AI;
	func_block.FIRE := FIRE;
	func_block.WIND := WIND ;
	func_block.ALARM := ALARM ;
	func_block.DOOR    := DOOR    ;
	func_block.RAIN := RAIN;
	func_block.ALARM_UP := ALARM_UP;
	func_block.WIND_UP := WIND_UP ;
	func_block.RAIN_UP := RAIN_UP ;

	func_block();
	QU  := func_block.QU;
	QD  := func_block.QD;
	STATUS  := func_block.STATUS;
	PO  := func_block.PO;
	AO  := func_block.AO;
END_PROGRAM

CONFIGURATION Config0
	RESOURCE Res0 ON PLC
		TASK task0(INTERVAL := T#20ms,PRIORITY := 0);
		PROGRAM instance0 WITH task0 : program0;
	END_RESOURCE
END_CONFIGURATION

(* ---- BLIND_SET.ST ---- *)
FUNCTION UDINT_TO_TIME2:TIME

	VAR_INPUT
		IN :	UDINT;
	END_VAR

	UDINT_TO_TIME2 := DINT_TO_TIME(UDINT_TO_DINT(IN));

END_FUNCTION

FUNCTION_BLOCK T_PLC_MS_block
	VAR_OUTPUT
		T_PLC_MS :	UDINT;
	END_VAR

	VAR_EXTERNAL
		PLC_TICKS_PER_SEC :	INT;
		PLC_SYS_TICK_CNT :	DINT;
	END_VAR

	VAR
		debug :	BOOL;(*Debug-Mode ON / OFF*)
		N :	INT;(*Debug-Faktor*)
		Offset :	UDINT;(*Debug-Offset*)
		temp :	DWORD := DWORD#1;(*Debug-Offset*)
		mode :	BOOL;(*modus*)
		faktor :	UDINT;(*Systemtakt-Faktor*)
		init :	BOOL;
		v_plc_ticks_per_sec :	UDINT;
		base :	UDINT := UDINT#1000;
	END_VAR

	IF init = FALSE THEN
		v_plc_ticks_per_sec := INT_TO_UDINT(PLC_TICKS_PER_SEC);
		IF v_plc_ticks_per_sec = UDINT#1024 THEN
			faktor := UDINT#1;
			mode := FALSE;
		ELSIF v_plc_ticks_per_sec > UDINT#0 THEN
			IF v_plc_ticks_per_sec <= base THEN
				faktor := base / v_plc_ticks_per_sec;
				mode := FALSE;
			ELSE
				faktor := v_plc_ticks_per_sec / base;
				mode := TRUE;
			END_IF;
		ELSE
			faktor := UDINT#1;
		END_IF;
		init := TRUE;
	END_IF;

	IF mode THEN
		T_PLC_MS := DINT_TO_UDINT(PLC_SYS_TICK_CNT) / faktor;
	ELSE
		T_PLC_MS := DINT_TO_UDINT(PLC_SYS_TICK_CNT) * faktor;
	END_IF;

	IF debug THEN
		T_PLC_MS := (DWORD_TO_UDINT(SHL(UDINT_TO_DWORD(T_PLC_MS),N) OR SHL(temp,N)) - UDINT#1) + Offset;
	END_IF;

END_FUNCTION_BLOCK

FUNCTION_BLOCK BLIND_SET_Block

	VAR_INPUT
		UP :	BOOL;
		DN :	BOOL;
		S_IN :	INT;
		PI :	BYTE;
		AI :	BYTE;
		IN :	BOOL;
		PX :	BYTE;
		AX :	BYTE;
		OVERRIDE_MANUAL :	BOOL;
		RESTORE_POSITION :	BOOL;
		RESTORE_TIME :	TIME := T#60s;
	END_VAR

	VAR_OUTPUT
		QU :	BOOL;
		QD :	BOOL;
		STATUS :	INT;
		PO :	BYTE;
		AO :	BYTE;
	END_VAR

	VAR
		T_PLC_MS :	T_PLC_MS_Block;
		tx :	TIME;
		ps :	BYTE;
		as :	BYTE;
		last :	TIME;
	END_VAR

	T_PLC_MS();
	tx:= UDINT_TO_TIME(T_PLC_MS.T_PLC_MS);

	IF IN THEN
		IF override_manual OR (UP AND DN) THEN
			status := 178;
		END_IF;
	END_IF;

	CASE STATUS OF
		0:
			status := S_IN;

		178:
			PO := PX;
			AO := AX;
			QU := TRUE;
			QD := TRUE;
			IF NOT in THEN
				STATUS := SEL(RESTORE_POSITION, S_IN, 179);
				last := tx;
			END_IF;

		179:
			PO := ps;
			AO := as;
			IF ((PO = PI) AND (AO = AI))  OR tx - last >= RESTORE_TIME THEN
				status := S_IN;
			END_IF;

	ELSE
		PO := PI;
		ps := PI;
		AO := AI;
		as := AI;
		STATUS := S_IN;
		QU := UP;
		QD := DN;
	END_CASE;

END_FUNCTION_BLOCK

PROGRAM program0
	VAR
		UP :	BOOL;
		DN :	BOOL;
		S_IN :	INT;
		PI :	BYTE;
		AI :	BYTE;
		IN :	BOOL;
		PX :	BYTE;
		AX :	BYTE;
		OVERRIDE_MANUAL :	BOOL;
		RESTORE_POSITION :	BOOL;
		RESTORE_TIME :	TIME := T#60s;
		QU :	BOOL;
		QD :	BOOL;
		STATUS :	INT;
		PO :	BYTE;
		AO :	BYTE;

		func_block : BLIND_SET_Block;
	END_VAR
	func_block.UP := UP;
	func_block.DN := DN;
	func_block.S_IN := S_IN ;
	func_block.PI    := PI    ;
	func_block.AI := AI;
	func_block.IN := IN;
	func_block.PX := PX ;
	func_block.AX := AX ;
	func_block.OVERRIDE_MANUAL    := OVERRIDE_MANUAL    ;
	func_block.RESTORE_POSITION := RESTORE_POSITION;
	func_block.RESTORE_TIME := RESTORE_TIME;

	func_block();
	QU  := func_block.QU;
	QD  := func_block.QD;
	STATUS  := func_block.STATUS;
	PO  := func_block.PO;
	AO  := func_block.AO;
END_PROGRAM

CONFIGURATION Config0
	VAR_GLOBAL
		PLC_TICKS_PER_SEC :	INT;
		PLC_SYS_TICK_CNT :	DINT;
	END_VAR
  	RESOURCE Res0 ON PLC
    	TASK task0(INTERVAL := T#20ms,PRIORITY := 0);
    	PROGRAM instance0 WITH task0 : program0;
  	END_RESOURCE
END_CONFIGURATION

(* ---- BLIND_SHADE_S.ST ---- *)
TYPE
  oscat_STRING5               : STRING;
  oscat_STRING30              : STRING;
END_TYPE

TYPE oscat_CALENDAR :
	STRUCT
		UTC : UDINT;				(* world time UTC *)
		LDT : UDINT;				(* local time *)
		LDATE : UDINT;				(* local date *)
		LTOD : UDINT;				(* local time of day *)
		YEAR : INT;					(* year of LDATE *)
		MONTH : INT;				(* month of LDATE *)
		DAY : INT;					(* day of LDATE *)
		WEEKDAY : INT;				(* weekday of LDATE *)
		OFFSET : INT;				(* Time Zone Offset for Local time in minutes *)
		DST_EN : BOOL;				(* daylight savings time enable *)
		DST_ON : BOOL;				(* true when daylight savings time os on *)
		NAME : oscat_string5;		(* name of time zone *)
		LANGUAGE : INT;			    (* language number pls see language setup *)
		LONGITUDE : REAL;			(* longitude of current location *)
		LATITUDE : REAL;			(* latitude of current location *)
		SUN_RISE : UDINT;			(* sun_rise for current location *)
		SUN_SET : UDINT;			(* sun_set for current location *)
		SUN_MIDDAY : UDINT;			(* worldtime when sun stands at south position *)
		SUN_HEIGTH : REAL;			(* suns heigth at midday, south position *)
		SUN_HOR : REAL;				(* sun angle horizontal 0 = north in degrees *)
		SUN_VER : REAL;				(* sun angle vertical above horizon in degrees *)
		NIGHT : BOOL;				(* true between sun_set and sun_rise *)
		HOLIDAY : BOOL;				(* true when holiday *)
		HOLY_NAME : oscat_string30;	(* name of holiday *)
		WORK_WEEK : INT;			(* current work week *)
	END_STRUCT;
END_TYPE

FUNCTION DT_TO_TOD2:UDINT
	VAR_INPUT
		IN :	UDINT;
	END_VAR

	DT_TO_TOD2 := (IN MOD UDINT#86400) * UDINT#1000;
END_FUNCTION

FUNCTION TIME_TO_UDINT2:UDINT
	VAR_INPUT
		X :	TIME;
	END_VAR

	TIME_TO_UDINT2 := DINT_TO_UDINT(TIME_TO_DINT(X));
END_FUNCTION

FUNCTION_BLOCK BLIND_SHADE_S_Block

	VAR_INPUT
		UP :	BOOL;
		DN :	BOOL;
		S_IN :	BYTE;
		PI :	BYTE;
		ENABLE :	BOOL;
		SUN :	BOOL;
		HORZ1 :	REAL := 100.0;
		HORZ2 :	REAL := 260.0;
		VERT :	REAL := 90.0;
		ALERT :	BOOL;
		SUNRISE_OFFSET :	TIME := T#1h;
		SUNSET_PRESET :	TIME := T#1h;
		SHADE_DELAY :	TIME := T#60s;
		SHADE_POS :	BYTE;
		QU :	BOOL;
		QD :	BOOL;
		STATUS :	BYTE;
		PO :	BYTE;
	END_VAR

	VAR_IN_OUT
		CX :	oscat_CALENDAR;
	END_VAR

	VAR
		angle :	REAL;
		sun_delay :	TOF;
	END_VAR

	sun_delay(IN := sun, PT := shade_delay);

	IF ALERT THEN
	QU := TRUE;
	QD := FALSE;
	STATUS := BYTE#152;
	ELSIF UP AND DN AND ENABLE AND sun_delay.Q
	AND (CX.SUN_HOR > HORZ1) AND (CX.SUN_HOR < HORZ2)
	AND (CX.SUN_VER < VERT)
	AND (DT_TO_TOD2(CX.UTC) > CX.SUN_RISE + TIME_TO_UDINT2(sunrise_offset)) AND (DT_TO_TOD2(CX.UTC) < CX.SUN_SET - TIME_TO_UDINT2(sunset_preset)) THEN
	QU := UP;
	QD := DN;
	STATUS := BYTE#151;
	PO := MIN(PI, shade_pos);
	ELSE
	QU := UP;
	QD := DN;
	PO := PI;
	STATUS := S_IN;
	END_IF;

END_FUNCTION_BLOCK

PROGRAM program0
	VAR
		UP :	BOOL;
		DN :	BOOL;
		S_IN :	BYTE;
		PI :	BYTE;
		ENABLE :	BOOL;
		SUN :	BOOL;
		HORZ1 :	REAL := 100.0;
		HORZ2 :	REAL := 260.0;
		VERT :	REAL := 90.0;
		ALERT :	BOOL;
		SUNRISE_OFFSET :	TIME := T#1h;
		SUNSET_PRESET :	TIME := T#1h;
		SHADE_DELAY :	TIME := T#60s;
		SHADE_POS :	BYTE;
		QU :	BOOL;
		QD :	BOOL;
		STATUS :	BYTE;
		PO :	BYTE;
		CX :	oscat_CALENDAR;

		func_block : BLIND_SHADE_S_Block;
	END_VAR
	func_block.UP := UP;
	func_block.DN := DN;
	func_block.S_IN := S_IN ;
	func_block.PI    := PI    ;
	func_block.ENABLE := ENABLE;
	func_block.SUN := SUN;
	func_block.HORZ1 := HORZ1 ;
	func_block.HORZ2 := HORZ2 ;
	func_block.VERT    := VERT    ;
	func_block.ALERT := ALERT;
	func_block.SUNRISE_OFFSET := SUNRISE_OFFSET;
	func_block.SUNSET_PRESET := SUNSET_PRESET ;
	func_block.SHADE_DELAY := SHADE_DELAY ;
	func_block.SHADE_POS    := SHADE_POS    ;
	func_block.QU := QU;
	func_block.QD := QD;
	func_block.STATUS := STATUS ;
	func_block.PO := PO ;
	func_block.CX := CX ;

	func_block();
	CX  := func_block.CX;
END_PROGRAM

CONFIGURATION Config0
	RESOURCE Res0 ON PLC
		TASK task0(INTERVAL := T#20ms,PRIORITY := 0);
		PROGRAM instance0 WITH task0 : program0;
	END_RESOURCE
END_CONFIGURATION

(* ---- BOILER.ST ---- *)
FUNCTION_BLOCK BOILER_Block

	VAR_INPUT
		T_UPPER :	REAL;
		T_LOWER :	REAL;
		PRESSURE :	BOOL := TRUE;
		ENABLE :	BOOL := TRUE;
		REQ_1 :	BOOL;
		REQ_2 :	BOOL;
		BOOST :	BOOL;
		T_UPPER_MIN :	REAL := REAL#50.0;
		T_UPPER_MAX :	REAL := REAL#60.0;
		T_LOWER_ENABLE :	BOOL;
		T_LOWER_MAX :	REAL := REAL#60.0;
		T_REQUEST_1 :	REAL := REAL#70.0;
		T_REQUEST_2 :	REAL := REAL#50.0;
		T_REQUEST_HYS :	REAL := REAL#5.0;
		T_PROTECT_HIGH :	REAL := REAL#80.0;
		T_PROTECT_LOW :	REAL := REAL#10.0;
	END_VAR

	VAR_OUTPUT
		HEAT :	BOOL;
		ERROR :	BOOL;
		STATUS :	BYTE;
	END_VAR

	VAR
		edge :	BOOL;
		boost_mode :	BOOL;
		flag_0 :	BOOL;
		flag_1 :	BOOL;
		flag_2 :	BOOL;
	END_VAR

	IF t_upper > t_protect_high THEN
		status := BYTE#1;
		heat := FALSE;
		error := TRUE;
	ELSIF t_upper < t_protect_low THEN
		status := BYTE#2;
		heat := TRUE;
		error := TRUE;
	ELSIF t_lower > T_protect_high AND t_lower_enable THEN
		status := BYTE#3;
		heat := FALSE;
		error := TRUE;
	ELSIF t_lower < t_protect_low AND t_lower_enable THEN
		status := BYTE#4;
		heat := TRUE;
		error := TRUE;
	ELSIF NOT pressure THEN
		status := BYTE#5;
		heat := FALSE;
		error := TRUE;
	ELSIF req_1 OR req_2 OR enable OR boost THEN
		error := FALSE;

		IF boost AND NOT edge AND t_upper < t_upper_max THEN
			status := BYTE#101;
			heat := TRUE;
			boost_mode := TRUE;
		ELSIF enable AND t_upper < T_upper_min THEN
			status := BYTE#102;
			heat := TRUE;
		ELSIF req_1 AND t_upper < T_request_1 THEN
			status := BYTE#103;
			heat := TRUE;
		ELSIF req_2 AND t_upper < t_request_2 THEN
			status := BYTE#104;
			heat := TRUE;
		END_IF;

		IF heat THEN
			IF (enable OR boost_mode) THEN
				flag_0 := TRUE;
				IF T_lower_enable AND T_lower > T_lower_max THEN
					flag_0 := FALSE;
					boost_mode := FALSE;
				ELSIF NOT T_lower_enable AND T_upper > T_upper_max THEN
					flag_0 := FALSE;
					boost_mode := FALSE;
				END_IF;
			ELSE
				flag_0 := FALSE;
			END_IF;
			flag_1 := (req_1 AND T_upper > T_request_1 + T_request_hys) AND req_1;
			flag_2 := (req_2 AND T_upper > T_request_2 + T_request_hys) AND req_2;

			heat := flag_0 OR flag_1 OR flag_2;
			IF heat = FALSE THEN status := BYTE#100; END_IF;
		END_IF;
	ELSE
		status := BYTE#100;
		heat := FALSE;
		error := FALSE;
	END_IF;
	edge := boost;

END_FUNCTION_BLOCK

PROGRAM program0
	VAR
		T_UPPER :	REAL;
		T_LOWER :	REAL;
		PRESSURE :	BOOL := TRUE;
		ENABLE :	BOOL := TRUE;
		REQ_1 :	BOOL;
		REQ_2 :	BOOL;
		BOOST :	BOOL;
		T_UPPER_MIN :	REAL := REAL#50.0;
		T_UPPER_MAX :	REAL := REAL#60.0;
		T_LOWER_ENABLE :	BOOL;
		T_LOWER_MAX :	REAL := REAL#60.0;
		T_REQUEST_1 :	REAL := REAL#70.0;
		T_REQUEST_2 :	REAL := REAL#50.0;
		T_REQUEST_HYS :	REAL := REAL#5.0;
		T_PROTECT_HIGH :	REAL := REAL#80.0;
		T_PROTECT_LOW :	REAL := REAL#10.0;
		HEAT :	BOOL;
		ERROR :	BOOL;
		STATUS :	BYTE;

		func_block : BOILER_Block;
	END_VAR
	func_block.T_UPPER := T_UPPER;
	func_block.T_LOWER := T_LOWER;
	func_block.PRESSURE := PRESSURE ;
	func_block.ENABLE    := ENABLE    ;
	func_block.REQ_1 := REQ_1;
	func_block.REQ_2 := REQ_2;
	func_block.BOOST := BOOST ;
	func_block.T_UPPER_MIN := T_UPPER_MIN ;
	func_block.T_UPPER_MAX    := T_UPPER_MAX    ;
	func_block.T_LOWER_ENABLE := T_LOWER_ENABLE;
	func_block.T_LOWER_MAX := T_LOWER_MAX;
	func_block.T_REQUEST_1 := T_REQUEST_1 ;
	func_block.T_REQUEST_2 := T_REQUEST_2 ;
	func_block.T_REQUEST_HYS    := T_REQUEST_HYS    ;
	func_block.T_PROTECT_HIGH := T_PROTECT_HIGH;
	func_block.T_PROTECT_LOW := T_PROTECT_LOW;

	func_block();
	HEAT  := func_block.HEAT;
	ERROR  := func_block.ERROR;
	STATUS  := func_block.STATUS;
END_PROGRAM

CONFIGURATION Config0
	RESOURCE Res0 ON PLC
		TASK task0(INTERVAL := T#20ms,PRIORITY := 0);
		PROGRAM instance0 WITH task0 : program0;
	END_RESOURCE
END_CONFIGURATION

(* ---- BUFFER_COMP.ST ---- *)
TYPE
	oscat_arb_0_249 			  : ARRAY [0..249] 	OF BYTE;
END_TYPE

FUNCTION_BLOCK BUFFER_COMP_Block
	VAR_IN_OUT
		PT1 :	oscat_arb_0_249;
	END_VAR

	VAR_INPUT
		SIZE1 :	INT;
	END_VAR

	VAR_IN_OUT
		PT2 :	oscat_arb_0_249;
	END_VAR

	VAR_INPUT
		SIZE2 :	INT;
		START :	INT;
	END_VAR

	VAR_OUTPUT
		BUFFER_COMP :	INT;
	END_VAR

	VAR
		i :	INT;
		j :	INT;
		end :	INT;
		j2 :	INT;
	END_VAR

	IF SIZE2 <= SIZE1 AND SIZE1 > 0 AND SIZE2 > 0 AND START >= 0 THEN
		end := SIZE1 - SIZE2;
		FOR i := START TO end DO
			IF PT1[i] = PT2[0] THEN
				(* first character matches, now compare rest of array *)
				j := 1;
				j2 := j + i;
				WHILE j < SIZE2 DO
					IF PT2[j] <> PT1[j2] THEN EXIT; END_IF;
					j := j + 1;
					j2 := j2 + 1;
				END_WHILE;
				(* when J > size2 a match was found return the position i in buffer1 *)
				IF j = SIZE2 THEN
					BUFFER_COMP := i;
					RETURN;
				END_IF;
			END_IF;
		END_FOR;
	END_IF;
	BUFFER_COMP := -1;

END_FUNCTION_BLOCK

PROGRAM program0
  VAR
    LocalVar0 : oscat_arb_0_249;
    LocalVar1 : INT;
	LocalVar2 : oscat_arb_0_249;
	LocalVar3 : INT;
	LocalVar4 : INT;
	LocalOUT  : INT;
	func_block : BUFFER_COMP_Block;
  END_VAR
	func_block.PT1  := LocalVar0;
	func_block.SIZE1 := LocalVar1;
	func_block.PT2  := LocalVar2;
	func_block.SIZE2 := LocalVar3;
	func_block.START := LocalVar4;
	func_block();
	LocalOUT := func_block.BUFFER_COMP;
	LocalVar0 := func_block.PT1;
	LocalVar2 := func_block.PT1;

END_PROGRAM

CONFIGURATION Config0
  RESOURCE Res0 ON PLC
    TASK task0(INTERVAL := T#20ms,PRIORITY := 0);
    PROGRAM instance0 WITH task0 : program0;
  END_RESOURCE
END_CONFIGURATION

(* ---- BUFFER_COMP_NW.ST ---- *)
TYPE
  oscat_NW_BUF_LONG  : ARRAY [0..4095] OF BYTE;
END_TYPE

FUNCTION_BLOCK BUFFER_COMP_NW
	VAR_IN_OUT
		PT1 :	oscat_NW_BUF_LONG;
	END_VAR

	VAR_INPUT
		SIZE1 :	INT;
	END_VAR

	VAR_IN_OUT
		PT2 :	oscat_NW_BUF_LONG;
	END_VAR

	VAR_INPUT
		SIZE2 :	INT;
		START :	INT;
	END_VAR

	VAR_OUTPUT
		BUFFER_COMP :	INT;
	END_VAR

	VAR
		i :	INT;
		j :	INT;
		end :	INT;
		j2 :	INT;
	END_VAR

	IF SIZE2 <= SIZE1 AND SIZE1 > 0 AND SIZE2 > 0 AND START >= 0 THEN
		end := SIZE1 - SIZE2;
		FOR i := START TO end DO
			IF PT1[i] = PT2[0] THEN
				(* first character matches, now compare rest of array *)
				j := 1;
				j2 := j + i;
				WHILE j < SIZE2 DO
					IF PT2[j] <> PT1[j2] THEN EXIT; END_IF;
					j := j + 1;
					j2 := j2 + 1;
				END_WHILE;
				(* when J > size2 a match was found return the position i in buffer1 *)
				IF j = SIZE2 THEN
					BUFFER_COMP := i;
					RETURN;
				END_IF;
			END_IF;
		END_FOR;
	END_IF;
	BUFFER_COMP := -1;

END_FUNCTION_BLOCK

PROGRAM program0
  VAR
	PT1   :	oscat_NW_BUF_LONG;

	SIZE1 :	INT;

	PT2   : 	oscat_NW_BUF_LONG;

	SIZE2 :	INT;
	START :	INT;

	BUFFER_COMP :	INT;

	func_block : BUFFER_COMP_NW;
  END_VAR
	func_block.PT1  :=PT1  ;
	func_block.SIZE1:=SIZE1;
	func_block.PT2  :=PT2  ;
	func_block.SIZE2:=SIZE2;
	func_block.START:=START;
	func_block();
	BUFFER_COMP := func_block.BUFFER_COMP;
	PT1 := func_block.PT1;
	PT2 := func_block.PT2;

END_PROGRAM

CONFIGURATION Config0
  RESOURCE Res0 ON PLC
    TASK task0(INTERVAL := T#20ms,PRIORITY := 0);
    PROGRAM instance0 WITH task0 : program0;
  END_RESOURCE
END_CONFIGURATION

(* ---- BYTE_TO_BITS.ST ---- *)
FUNCTION BIT_OF_DWORD : BOOL
  VAR_INPUT
    IN : DWORD;
    N : INT;
  END_VAR

  BIT_OF_DWORD := (SHR(in,N) AND 16#00000001) > 0;
END_FUNCTION

FUNCTION_BLOCK BYTE_TO_BITS
	VAR_INPUT
		IN :	BYTE;
	END_VAR

	VAR_OUTPUT
		B0 :	BOOL;
		B1 :	BOOL;
		B2 :	BOOL;
		B3 :	BOOL;
		B4 :	BOOL;
		B5 :	BOOL;
		B6 :	BOOL;
		B7 :	BOOL;
	END_VAR

	B0 := BIT_OF_DWORD(BYTE_TO_DWORD(IN),0); (* IN.X0 *)
	B1 := BIT_OF_DWORD(BYTE_TO_DWORD(IN),1); (* IN.X1 *)
	B2 := BIT_OF_DWORD(BYTE_TO_DWORD(IN),2); (* IN.X2 *)
	B3 := BIT_OF_DWORD(BYTE_TO_DWORD(IN),3); (* IN.X3 *)
	B4 := BIT_OF_DWORD(BYTE_TO_DWORD(IN),4); (* IN.X4 *)
	B5 := BIT_OF_DWORD(BYTE_TO_DWORD(IN),5); (* IN.X5 *)
	B6 := BIT_OF_DWORD(BYTE_TO_DWORD(IN),6); (* IN.X6 *)
	B7 := BIT_OF_DWORD(BYTE_TO_DWORD(IN),7); (* IN.X7 *)
END_FUNCTION_BLOCK

PROGRAM program0
  VAR
	LocalVar0  : BYTE;
	B0 :	BOOL;
	B1 :	BOOL;
	B2 :	BOOL;
	B3 :	BOOL;
	B4 :	BOOL;
	B5 :	BOOL;
	B6 :	BOOL;
	B7 :	BOOL;
	func_block: BYTE_TO_BITS;
  END_VAR

	func_block.IN  := LocalVar0;
	func_block();
	B0 := func_block.B0;
	B1 := func_block.B1;
	B2 := func_block.B2;
	B3 := func_block.B3;
	B4 := func_block.B4;
	B5 := func_block.B5;
	B6 := func_block.B6;
	B7 := func_block.B7;

END_PROGRAM

CONFIGURATION Config0
  RESOURCE Res0 ON PLC
    TASK task0(INTERVAL := T#20ms,PRIORITY := 0);
    PROGRAM instance0 WITH task0 : program0;
  END_RESOURCE
END_CONFIGURATION

(* ---- BYTE_TO_STRB.ST ---- *)
FUNCTION_BLOCK BYTE_TO_STRB_Block
	VAR_INPUT
		IN :	BYTE;
	END_VAR

	VAR_OUTPUT
		BYTE_TO_STRB :	STRING;
	END_VAR

	VAR
		i :	INT;
	END_VAR

	BYTE_TO_STRB := '';
	FOR i := 1 TO 8 DO
		IF (in AND BYTE#2#1000_0000) = BYTE#2#1000_0000 THEN
			BYTE_TO_STRB := CONCAT(BYTE_TO_STRB,'1');
		ELSE
			BYTE_TO_STRB := CONCAT(BYTE_TO_STRB,'0');
		END_IF;
		in := SHL(in, 1);
	END_FOR;

END_FUNCTION_BLOCK

PROGRAM program0
  VAR
    LocalVar0 : BYTE;
	LocalOUT  : STRING;
	func_block : BYTE_TO_STRB_Block;
  END_VAR
	func_block.IN  := LocalVar0;
	func_block();
	LocalOUT := func_block.BYTE_TO_STRB;

END_PROGRAM

CONFIGURATION Config0
  RESOURCE Res0 ON PLC
    TASK task0(INTERVAL := T#20ms,PRIORITY := 0);
    PROGRAM instance0 WITH task0 : program0;
  END_RESOURCE
END_CONFIGURATION

(* ---- BYTE_TO_STRH.ST ---- *)
FUNCTION_BLOCK BYTE_TO_STRH_Block
	VAR_INPUT
		IN :	BYTE;
	END_VAR

	VAR_OUTPUT
		BYTE_TO_STRH :	STRING;
	END_VAR

	BYTE_TO_STRH:=BYTE_TO_STRING(IN);

END_FUNCTION_BLOCK

PROGRAM program0
  VAR
    LocalVar0 : BYTE;
	LocalOUT  : STRING;
	func_block : BYTE_TO_STRH_Block;
  END_VAR
	func_block.IN  := LocalVar0;
	func_block();
	LocalOUT := func_block.BYTE_TO_STRH;

END_PROGRAM

CONFIGURATION Config0
  RESOURCE Res0 ON PLC
    TASK task0(INTERVAL := T#20ms,PRIORITY := 0);
    PROGRAM instance0 WITH task0 : program0;
  END_RESOURCE
END_CONFIGURATION

(* ---- CABS.ST ---- *)
TYPE oscat_complex :
  STRUCT
	re : REAL;
	im : REAL;
  END_STRUCT;
END_TYPE

FUNCTION HYPOT:REAL
	VAR_INPUT
		X :	REAL;
		Y :	REAL;
	END_VAR

	HYPOT := SQRT(x*x + y*y);
END_FUNCTION

FUNCTION_BLOCK CABS_Block
	VAR_INPUT
		X :	oscat_complex;
	END_VAR

	VAR_OUTPUT
		CABS :	REAL;
	END_VAR

	CABS := HYPOT(x.re, x.im);

END_FUNCTION_BLOCK

PROGRAM program0
  VAR
    LocalVar0 : oscat_complex;
	LocalOUT  : REAL;
	func_block : CABS_Block;
  END_VAR
	func_block.X  := LocalVar0;
	func_block();
	LocalOUT := func_block.CABS;

END_PROGRAM

CONFIGURATION Config0
  RESOURCE Res0 ON PLC
    TASK task0(INTERVAL := T#20ms,PRIORITY := 0);
    PROGRAM instance0 WITH task0 : program0;
  END_RESOURCE
END_CONFIGURATION

(* ---- CACOS.ST ---- *)
TYPE oscat_complex :
  STRUCT
	re : REAL;
	im : REAL;
  END_STRUCT;
END_TYPE

FUNCTION ATAN2:REAL
	VAR_INPUT
		X :	REAL;
		Y :	REAL;
	END_VAR

	IF X > 0.0 THEN
		ATAN2 := ATAN(Y/X);
	ELSIF X < 0.0 THEN
		IF Y >= 0.0 THEN
			ATAN2 := ATAN(Y/X) + 3.14159265358979323846264338327950288;
		ELSE
			ATAN2 := ATAN(Y/X) - 3.14159265358979323846264338327950288;
		END_IF;
	ELSIF Y > 0.0 THEN
		ATAN2 := 1.5707963267948965580;
	ELSIF Y < 0.0 THEN
		ATAN2 := -1.5707963267948965580;
	ELSE
		ATAN2 := 0.0;
	END_IF;

END_FUNCTION

FUNCTION HYPOT:REAL
	VAR_INPUT
		X :	REAL;
		Y :	REAL;
	END_VAR

	HYPOT := SQRT(x*x + y*y);
END_FUNCTION

FUNCTION_BLOCK CLOG_Block

	VAR_INPUT
		X :	oscat_complex;
	END_VAR

	VAR_OUTPUT
		CLOG :	oscat_complex;
	END_VAR

	CLOG.re := LN(HYPOT(X.re, X.im));
	CLOG.im := ATAN2(X.im, X.re);

END_FUNCTION_BLOCK

FUNCTION SGN : INT
  VAR_INPUT
    x : REAL;
  END_VAR

  IF X > 0.0 THEN
  	sgn := 1;
  ELSIF X < 0.0 THEN
  	sgn := -1;
  ELSE
  	sgn := 0;
  END_IF;
END_FUNCTION

FUNCTION_BLOCK CSQRT_Block
	VAR_INPUT
		X :	oscat_complex;
	END_VAR

	VAR_OUTPUT
		CSQRT :	oscat_complex;
	END_VAR

	VAR
		temp :	REAL;
	END_VAR

	temp := HYPOT(x.re, x.im);
	CSQRT.re :=  SQRT(0.5 * (temp + x.re));
	CSQRT.im :=  INT_TO_REAL(sgn(x.im)) * SQRT(0.5 * (temp - x.re));

END_FUNCTION_BLOCK

FUNCTION_BLOCK CACOSH_Block
	VAR_INPUT
		X :	oscat_complex;
	END_VAR

	VAR_OUTPUT
		CACOSH :	oscat_complex;
	END_VAR

	VAR
		Y :	oscat_complex;
		CLOG :	CLOG_Block;
		CSQRT :	CSQRT_Block;
	END_VAR

	y.re := (X.re - X.im)*(X.re + X.im) - 1.0;
	y.im := 2.0 * X.re * X.im;
	CSQRT(X:=y);
	y    := CSQRT.CSQRT;
	y.re := y.re + x.re;
	y.im := y.im + x.im;
	CLOG(X:=y);
	CACOSH  := CLOG.CLOG;
END_FUNCTION_BLOCK

FUNCTION_BLOCK CACOS_Block
	VAR_INPUT
		X :	oscat_complex;
	END_VAR

	VAR_OUTPUT
		CACOS :	oscat_complex;
	END_VAR

	VAR
		Y :	oscat_complex;
		CACOSH :	CACOSH_Block;
	END_VAR

	CACOSH(X:=x);
	y := CACOSH.CACOSH;
	CACOS.re := y.im;
	CACOS.im := -y.re;
END_FUNCTION_BLOCK

PROGRAM program0
  VAR
    LocalVar0 : oscat_complex;
	LocalOUT  : oscat_complex;
	func_block : CACOS_Block;
  END_VAR
	func_block.X  := LocalVar0;
	func_block();
	LocalOUT := func_block.CACOS;
END_PROGRAM

CONFIGURATION Config0
  RESOURCE Res0 ON PLC
    TASK task0(INTERVAL := T#20ms,PRIORITY := 0);
    PROGRAM instance0 WITH task0 : program0;
  END_RESOURCE
END_CONFIGURATION

(* ---- CACOSH.ST ---- *)
TYPE oscat_complex :
  STRUCT
	re : REAL;
	im : REAL;
  END_STRUCT;
END_TYPE

FUNCTION ATAN2:REAL
	VAR_INPUT
		X :	REAL;
		Y :	REAL;
	END_VAR

	IF X > 0.0 THEN
		ATAN2 := ATAN(Y/X);
	ELSIF X < 0.0 THEN
		IF Y >= 0.0 THEN
			ATAN2 := ATAN(Y/X) + 3.14159265358979323846264338327950288;
		ELSE
			ATAN2 := ATAN(Y/X) - 3.14159265358979323846264338327950288;
		END_IF;
	ELSIF Y > 0.0 THEN
		ATAN2 := 1.5707963267948965580;
	ELSIF Y < 0.0 THEN
		ATAN2 := -1.5707963267948965580;
	ELSE
		ATAN2 := 0.0;
	END_IF;

END_FUNCTION

FUNCTION HYPOT:REAL
	VAR_INPUT
		X :	REAL;
		Y :	REAL;
	END_VAR

	HYPOT := SQRT(x*x + y*y);
END_FUNCTION

FUNCTION_BLOCK CLOG_Block

	VAR_INPUT
		X :	oscat_complex;
	END_VAR

	VAR_OUTPUT
		CLOG :	oscat_complex;
	END_VAR

	CLOG.re := LN(HYPOT(X.re, X.im));
	CLOG.im := ATAN2(X.im, X.re);

END_FUNCTION_BLOCK

FUNCTION SGN : INT
  VAR_INPUT
    x : REAL;
  END_VAR

  IF X > 0.0 THEN
  	sgn := 1;
  ELSIF X < 0.0 THEN
  	sgn := -1;
  ELSE
  	sgn := 0;
  END_IF;
END_FUNCTION

FUNCTION_BLOCK CSQRT_Block
	VAR_INPUT
		X :	oscat_complex;
	END_VAR

	VAR_OUTPUT
		CSQRT :	oscat_complex;
	END_VAR

	VAR
		temp :	REAL;
	END_VAR

	temp := HYPOT(x.re, x.im);
	CSQRT.re :=  SQRT(0.5 * (temp + x.re));
	CSQRT.im :=  INT_TO_REAL(sgn(x.im)) * SQRT(0.5 * (temp - x.re));

END_FUNCTION_BLOCK

FUNCTION_BLOCK CACOSH_Block
	VAR_INPUT
		X :	oscat_complex;
	END_VAR

	VAR_OUTPUT
		CACOSH :	oscat_complex;
	END_VAR

	VAR
		Y :	oscat_complex;
		CLOG :	CLOG_Block;
		CSQRT :	CSQRT_Block;
	END_VAR

	y.re := (X.re - X.im)*(X.re + X.im) - 1.0;
	y.im := 2.0 * X.re * X.im;
	CSQRT(X:=y);
	y    := CSQRT.CSQRT;
	y.re := y.re + x.re;
	y.im := y.im + x.im;
	CLOG(X:=y);
	CACOSH  := CLOG.CLOG;
END_FUNCTION_BLOCK

PROGRAM program0
  VAR
    LocalVar0 : oscat_complex;
	LocalOUT  : oscat_complex;
	func_block : CACOSH_Block;
  END_VAR
	func_block.X  := LocalVar0;
	func_block();
	LocalOUT := func_block.CACOSH;
END_PROGRAM

CONFIGURATION Config0
  RESOURCE Res0 ON PLC
    TASK task0(INTERVAL := T#20ms,PRIORITY := 0);
    PROGRAM instance0 WITH task0 : program0;
  END_RESOURCE
END_CONFIGURATION

(* ---- CADD.ST ---- *)
TYPE oscat_complex :
  STRUCT
	re : REAL;
	im : REAL;
  END_STRUCT;
END_TYPE

FUNCTION_BLOCK CADD_Block

	VAR_INPUT
		X :	oscat_complex;
		Y :	oscat_complex;
	END_VAR

	VAR_OUTPUT
		CADD :	oscat_complex;
	END_VAR

	CADD.re := x.re + y.re;
	CADD.im := x.im + y.im;

END_FUNCTION_BLOCK

PROGRAM program0
  VAR
    LocalVar0 : oscat_complex;
	LocalVar1 : oscat_complex;
	LocalOUT  : oscat_complex;
	func_block : CADD_Block;
  END_VAR
	func_block.X  := LocalVar0;
	func_block.Y  := LocalVar0;
	func_block();
	LocalOUT := func_block.CADD;
END_PROGRAM

CONFIGURATION Config0
  RESOURCE Res0 ON PLC
    TASK task0(INTERVAL := T#20ms,PRIORITY := 0);
    PROGRAM instance0 WITH task0 : program0;
  END_RESOURCE
END_CONFIGURATION

(* ---- CALENDAR_CALC.ST ---- *)
TYPE oscat_CALENDAR :
	STRUCT
		UTC : UDINT;				(* world time UTC *)
		LDT : UDINT;				(* local time *)
		LDATE : UDINT;				(* local date *)
		LTOD : UDINT;				(* local time of day *)
		YEAR : INT;					(* year of LDATE *)
		MONTH : INT;				(* month of LDATE *)
		DAY : INT;					(* day of LDATE *)
		WEEKDAY : INT;				(* weekday of LDATE *)
		OFFSET : INT;				(* Time Zone Offset for Local time in minutes *)
		DST_EN : BOOL;				(* daylight savings time enable *)
		DST_ON : BOOL;				(* true when daylight savings time os on *)
		NAME : STRING;		(* name of time zone *)
		LANGUAGE : INT;			    (* language number pls see language setup *)
		LONGITUDE : REAL;			(* longitude of current location *)
		LATITUDE : REAL;			(* latitude of current location *)
		SUN_RISE : UDINT;			(* sun_rise for current location *)
		SUN_SET : UDINT;			(* sun_set for current location *)
		SUN_MIDDAY : UDINT;			(* worldtime when sun stands at south position *)
		SUN_HEIGTH : REAL;			(* suns heigth at midday, south position *)
		SUN_HOR : REAL;				(* sun angle horizontal 0 = north in degrees *)
		SUN_VER : REAL;				(* sun angle vertical above horizon in degrees *)
		NIGHT : BOOL;				(* true between sun_set and sun_rise *)
		HOLIDAY : BOOL;				(* true when holiday *)
		HOLY_NAME : STRING;	(* name of holiday *)
		WORK_WEEK : INT;			(* current work week *)
	END_STRUCT;
END_TYPE

TYPE oscat_LANGUAGE:
  STRUCT
    DEFAULT 	: INT;
	LMAX    	: INT;
  END_STRUCT;
END_TYPE

TYPE
	oscat_LOCATION_ELEMENTS	: ARRAY [1..5] OF INT;
END_TYPE

TYPE
  oscat_ELEMENT_WEEKDAYS	: ARRAY [1..7] OF STRING;
  oscat_WEEKDAYS			: ARRAY [1..3]  OF oscat_ELEMENT_WEEKDAYS := [0, 0, 0];
END_TYPE

TYPE oscat_LOCATION:
  STRUCT
    DEFAULT 	: INT;
	LMAX    	: INT;
	LANGUAGE	: oscat_LOCATION_ELEMENTS;
  END_STRUCT;
END_TYPE

TYPE oscat_HOLIDAY_DATA :
  STRUCT
	NAME : STRING;
	DAY : SINT;
	MONTH : SINT;
	USE : SINT;
	PAD_BYTE : BYTE;
  END_STRUCT;
END_TYPE

TYPE
  oscat_HOLIDAY_DATA_0_29 	: ARRAY [0..29] OF oscat_HOLIDAY_DATA;
  oscat_HOLIDAY_DATA_0_49 	: ARRAY [0..49] OF oscat_HOLIDAY_DATA;
END_TYPE

FUNCTION _REAL_TO_UDINT:UDINT

	VAR_INPUT
		X :	REAL;
	END_VAR

	IF REAL_TO_UDINT(0.5) = UDINT#1 THEN
		_REAL_TO_UDINT := REAL_TO_UDINT(x);
	ELSIF X > 0.0 THEN
		_REAL_TO_UDINT := REAL_TO_UDINT(x+0.5);
	ELSIF X < 0.0 THEN
		_REAL_TO_UDINT := REAL_TO_UDINT(x-0.5);
	ELSE
		_REAL_TO_UDINT := UDINT#0;
  	END_IF;
END_FUNCTION

FUNCTION HOUR_TO_TIME:TIME

	VAR_INPUT
		IN :	REAL;
	END_VAR

	hour_to_time := UDINT_TO_TIME(_REAL_TO_UDINT(IN * 3600000.0));
END_FUNCTION

FUNCTION TIME_TO_UDINT2:UDINT
	VAR_INPUT
		X :	TIME;
	END_VAR

	TIME_TO_UDINT2 := DINT_TO_UDINT(TIME_TO_DINT(X));
END_FUNCTION

FUNCTION FLOOR2 : DINT
	VAR_INPUT
		x : REAL;
	END_VAR

	FLOOR2 := REAL_TO_DINT(X);
	IF DINT_TO_REAL(FLOOR2) > X THEN
		FLOOR2 := FLOOR2 - DINT#1;
	END_IF;

END_FUNCTION

FUNCTION MODR:REAL

	VAR_INPUT
		IN :	REAL;
		DIVI :	REAL;
	END_VAR

	IF divi = 0.0 THEN
		MODR := 0.0;
	ELSE
		MODR := in - DINT_TO_REAL(FLOOR2(in / divi)) * divi;
	END_IF;

END_FUNCTION

FUNCTION RAD:REAL

	VAR_INPUT
		DEGG :	REAL;
	END_VAR

	RAD := MODR(0.0174532925199433 * DEGG , 6.283185307179586476);

END_FUNCTION

FUNCTION REFRACTION:REAL

	VAR_INPUT
		ELEV :	REAL;
	END_VAR

	VAR
		tmp :	REAL;
	END_VAR

	tmp := LIMIT(-1.9, elev, 80.0);
	REFRACTION := 0.0174532925199433 / TAN(0.0174532925199433 * (tmp + 10.3 / (tmp + 5.11)));

END_FUNCTION

FUNCTION TOD_TO_REAL2:REAL
	VAR_INPUT
		IN :	UDINT;
	END_VAR
	TOD_TO_REAL2 := UDINT_TO_REAL(IN);
END_FUNCTION

FUNCTION DEG:REAL

	VAR_INPUT
		X :	REAL;
	END_VAR

	DEG := MODR(57.29577951308232 * X, 360.0);
END_FUNCTION

FUNCTION DT_TO_TOD2:UDINT
	VAR_INPUT
		IN :	UDINT;
	END_VAR

	DT_TO_TOD2 := (IN MOD UDINT#86400) * UDINT#1000;
END_FUNCTION

FUNCTION_BLOCK SUN_POS

	VAR_INPUT
		LATITUDE :	REAL;
		LONGITUDE :	REAL;
		UTC :	UDINT;
	END_VAR

	VAR_OUTPUT
		B :	REAL;
		HR :	REAL;
	END_VAR

	VAR
		g :	REAL;
		a :	REAL;
		d :	REAL;
		h :	REAL;
		t1 :	REAL;
		n :	REAL;
		e :	REAL;
		c :	REAL;
		tau :	REAL;
		sin_d :	REAL;
		rlat :	REAL;
		sin_lat :	REAL;
		cos_lat :	REAL;
		cos_tau :	REAL;
		cos_d :	REAL;
		MATH_PI :	REAL := 3.14159265358979323846264338327950288;
		MATH_PI2 :	REAL := 6.28318530717958647692528676655900576;
	END_VAR

	n := UDINT_TO_REAL(UTC - UDINT#946728000) * 0.000011574074074074;
	g :=MODR(6.240040768 + 0.01720197 * n, MATH_PI2);
	d := MODR(4.89495042 + 0.017202792 * n, MATH_PI2) + 0.033423055 * SIN(g) + 0.000349066 * SIN(2.0*g);
	e := 0.409087723 - 0.000000006981317008 * n;
	cos_d := COS(d);
	sin_d := SIN(d);
	a := ATAN(COS(e) * sin_d / cos_d);
	IF cos_d < 0.0 THEN a := a + MATH_PI; END_IF;
	c := ASIN(SIN(e) * sin_d);

	(* also here we must be very careful utc is from 1.1.1970 for step7 the formula must change *)
	tau := RAD(MODR(6.697376 + (n - 0.25) * 0.0657098245037645 + TOD_TO_REAL2(DT_TO_TOD2(utc)) * 0.0000002785383333, 24.0) * 15.0 + longitude) - a;
	rlat := RAD(latitude);
	sin_lat := SIN(rlat);
	cos_lat := COS(rlat);
	cos_tau := COS(tau);
	t1 := cos_tau * sin_lat - TAN(c) * cos_lat;
	B := ATAN(SIN(tau) / t1);
	IF t1 < 0.0 THEN B := B + MATH_PI2; ELSE B := B + MATH_PI; END_IF;
	B := DEG(MODR(B, MATH_PI2));
	h := DEG(ASIN(COS(C) * cos_tau * cos_lat +SIN(c) * sin_lat));
	IF h > 180.0 THEN h := h - 360.0; END_IF;
	(* consider refraction *)
	HR := h + REFRACTION(h);
END_FUNCTION_BLOCK

FUNCTION HOUR_TO_TOD:UDINT
	VAR_INPUT
		IN :	REAL;
	END_VAR

	hour_to_tod := _REAL_TO_UDINT(IN * 3600000.00);
END_FUNCTION

FUNCTION DAY_OF_YEAR:INT
	VAR_INPUT
		IDATE :	DATE;
	END_VAR

	DAY_OF_YEAR := UDINT_TO_INT((DATE_TO_UDINT(idate) / UDINT#86400) MOD UDINT#1461);
	IF DAY_OF_YEAR > 729 THEN
		IF DAY_OF_YEAR > 1095 THEN DAY_OF_YEAR := DAY_OF_YEAR - 1095; ELSE DAY_OF_YEAR := DAY_OF_YEAR - 729; END_IF;
	ELSIF DAY_OF_YEAR > 364 THEN
		DAY_OF_YEAR := DAY_OF_YEAR - 364;
	ELSE
		DAY_OF_YEAR := DAY_OF_YEAR + 1;
	END_IF;
END_FUNCTION

FUNCTION DAY_OF_YEAR_UDINT:INT
	VAR_INPUT
		IDATE :	UDINT;
	END_VAR

	DAY_OF_YEAR_UDINT := UDINT_TO_INT((idate / UDINT#86400) MOD UDINT#1461);
	IF DAY_OF_YEAR_UDINT > 729 THEN
		IF DAY_OF_YEAR_UDINT > 1095 THEN DAY_OF_YEAR_UDINT := DAY_OF_YEAR_UDINT - 1095; ELSE DAY_OF_YEAR_UDINT := DAY_OF_YEAR_UDINT - 729; END_IF;
	ELSIF DAY_OF_YEAR_UDINT > 364 THEN
		DAY_OF_YEAR_UDINT := DAY_OF_YEAR_UDINT - 364;
	ELSE
		DAY_OF_YEAR_UDINT := DAY_OF_YEAR_UDINT + 1;
	END_IF;
END_FUNCTION

FUNCTION SUN_MIDDAY:UDINT
	VAR_INPUT
		LON :	REAL;
		UTC :	DATE;
	END_VAR

	VAR
		T :	REAL;
		OFFSET :	REAL;
	END_VAR

	T := INT_TO_REAL(DAY_OF_YEAR(utc));
	OFFSET := -0.1752 * SIN(0.033430 * T + 0.5474) - 0.1340 * SIN(0.018234 * T - 0.1939);
	SUN_MIDDAY := HOUR_TO_TOD(12.0 - OFFSET - lon * 0.0666666666666);
END_FUNCTION

FUNCTION SUN_MIDDAY_UDINT:UDINT
	VAR_INPUT
		LON :	REAL;
		UTC :	UDINT;
	END_VAR

	VAR
		T :	REAL;
		OFFSET :	REAL;
	END_VAR

	T := INT_TO_REAL(DAY_OF_YEAR_UDINT(utc));
	OFFSET := -0.1752 * SIN(0.033430 * T + 0.5474) - 0.1340 * SIN(0.018234 * T - 0.1939);
	SUN_MIDDAY_UDINT := HOUR_TO_TOD(12.0 - OFFSET - lon * 0.0666666666666);
END_FUNCTION

FUNCTION_BLOCK SUN_TIME_Block

	VAR_INPUT
		LATITUDE :	REAL;
		LONGITUDE :	REAL;
		UTC :	UDINT;
		H :	REAL := -0.83333333333;
	END_VAR

	VAR_OUTPUT
		MIDDAY :	UDINT;
		SUN_RISE :	UDINT;
		SUN_SET :	UDINT;
		SUN_DECLINATION :	REAL;
	END_VAR

	VAR
		DK :	REAL;
		delta :	UDINT;
		B :	REAL;
	END_VAR

	B := latitude * 0.0174532925199433;
	MIDDAY := SUN_MIDDAY_UDINT(longitude, utc);
	DK := 0.40954 * SIN(0.0172 * (INT_TO_REAL(DAY_OF_YEAR_UDINT(utc)) - 79.35));
	sun_declination := DEG(DK);
	IF sun_declination > 180.0 THEN sun_declination := sun_declination - 360.0; END_IF;
	sun_declination := 90.0 - LATITUDE + sun_declination;
	delta := TIME_TO_UDINT2(HOUR_TO_TIME(ACOS((SIN(RAD(H)) - SIN(B) * SIN(DK)) / (COS(B) * COS(DK))) * 3.819718632));
	sun_rise := MIDDAY - delta;
	sun_set := MIDDAY + delta;
END_FUNCTION_BLOCK

FUNCTION_BLOCK SETUP_LANGUAGE_Block

	VAR_IN_OUT
		LANGUAGE :	oscat_LANGUAGE;
	END_VAR

	VAR
		init :	BOOL;
	END_VAR

	IF init THEN RETURN; END_IF;
	init := TRUE;

	LANGUAGE.DEFAULT  := 1; (* 1=english, 2=german 3=french *)
	LANGUAGE.LMAX := 3;
END_FUNCTION_BLOCK

FUNCTION_BLOCK SETUP_LOCATION
	VAR_IN_OUT
		LOCATION :	oscat_LOCATION;
	END_VAR

	VAR
		init :	BOOL;
	END_VAR

	IF init THEN RETURN; END_IF;
	init := TRUE;

	LOCATION.DEFAULT  := 1;
	LOCATION.LMAX := 5;

	LOCATION.LANGUAGE[1] := 2;
	LOCATION.LANGUAGE[2] := 2;
	LOCATION.LANGUAGE[3] := 3;
	LOCATION.LANGUAGE[4] := 2;
	LOCATION.LANGUAGE[5] := 2;
END_FUNCTION_BLOCK

FUNCTION_BLOCK SETUP_WEEKDAYS

	VAR_IN_OUT
		WEEKDAYS :	oscat_WEEKDAYS;
	END_VAR

	VAR
		init :	BOOL;
	END_VAR

	IF init THEN RETURN; END_IF;
	init := TRUE;

	WEEKDAYS[1][01] := 'Monday';
	WEEKDAYS[1][02] := 'Tuesday';
	WEEKDAYS[1][03] := 'Wednesday';
	WEEKDAYS[1][04] := 'Thursday';
	WEEKDAYS[1][05] := 'Friday';
	WEEKDAYS[1][06] := 'Saturday';
	WEEKDAYS[1][07] := 'Sunday';

	WEEKDAYS[2][01] := 'Montag';
	WEEKDAYS[2][02] := 'Dienstag';
	WEEKDAYS[2][03] := 'Mittwoch';
	WEEKDAYS[2][04] := 'Donnerstag';
	WEEKDAYS[2][05] := 'Freitag';
	WEEKDAYS[2][06] := 'Samstag';
	WEEKDAYS[2][07] := 'Sonntag';

	WEEKDAYS[3][01] := 'Lundi';
	WEEKDAYS[3][02] := 'Mardi';
	WEEKDAYS[3][03] := 'Mercredi';
	WEEKDAYS[3][04] := 'Jeudi';
	WEEKDAYS[3][05] := 'Vendredi';
	WEEKDAYS[3][06] := 'Samedi';
	WEEKDAYS[3][07] := 'Dimanche';
END_FUNCTION_BLOCK

FUNCTION YEAR_OF_DATE:INT
	VAR_INPUT
		IDATE :	UDINT;
	END_VAR

	YEAR_OF_DATE := UDINT_TO_INT((idate+UDINT#43200) / UDINT#31557600 + UDINT#1970);
END_FUNCTION

FUNCTION _INT_TO_UDINT:UDINT
	VAR_INPUT
		IN :	INT;
	END_VAR

	_INT_TO_UDINT := DINT_TO_UDINT(INT_TO_DINT(IN));
END_FUNCTION

FUNCTION SET_DATE:UDINT

	VAR_INPUT
		YEAR :	INT;
		MONTH :	INT;
		DAY :	INT;
	END_VAR

	VAR
		count :	INT;
	END_VAR

	IF month > 2 THEN
		count := (month - 1) * 30;
		IF month > 7 THEN
			count := count + DWORD_TO_INT(SHR(DINT_TO_DWORD(INT_TO_DINT(month) - INT_TO_DINT(3)),1));
		ELSE
			count := count + DWORD_TO_INT(SHR(DINT_TO_DWORD(INT_TO_DINT(month) - INT_TO_DINT(4)),1));
		END_IF;
		IF SHL(INT_TO_WORD(year),14) = WORD#0 THEN
			count := count + 1;
		END_IF;
	ELSE
		count := (month - 1) * 31;
	END_IF;
	SET_DATE := (_INT_TO_UDINT(count + day - 1) + DWORD_TO_UDINT(SHR(UDINT_TO_DWORD(_INT_TO_UDINT(year) * UDINT#1461 - UDINT#2878169), 2))) * UDINT#86400;
END_FUNCTION

FUNCTION DAY_OF_WEEK:INT
	VAR_INPUT
		IDATE :	UDINT;
	END_VAR

	DAY_OF_WEEK := UDINT_TO_INT((idate / UDINT#86400 + UDINT#3) MOD UDINT#7) + INT#01;
END_FUNCTION

FUNCTION EASTER:UDINT
	VAR_INPUT
		YEAR :	INT;
	END_VAR

	VAR
		b :	INT;
		c :	INT;
		oday :	INT;
	END_VAR

	b := (204 - 11 * (year MOD 19)) MOD 30;
	IF b > 27 THEN b := b - 1; END_IF;
	c := (year + WORD_TO_INT(SHR(INT_TO_WORD(year),2)) + b - 13) MOD 7;
	oday := 28 + b - c;
	IF oday > 33 THEN
		easter := set_Date(year, 4, oday - 31);
	ELSE
		easter := set_Date(year, 3, oday);
	END_IF;
END_FUNCTION

FUNCTION LEAP_OF_DATE:BOOL

	VAR_INPUT
		IDATE :	UDINT;
	END_VAR

	LEAP_OF_DATE := SHL(UDINT_TO_DWORD((idate + UDINT#43200) / UDINT#31557600), 30) = DWORD#16#80000000;
END_FUNCTION

FUNCTION MONTH_OF_DATE:INT

	VAR_INPUT
		IDATE :	UDINT;
	END_VAR

	MONTH_OF_DATE := DAY_OF_YEAR_UDINT(idate);
	IF MONTH_OF_DATE < 32 THEN
		MONTH_OF_DATE := 1;
	ELSIF LEAP_OF_DATE((IDATE)) THEN
		MONTH_OF_DATE := (MONTH_OF_DATE * 53 + 1668) / 1623;
	ELSE
		MONTH_OF_DATE := (MONTH_OF_DATE * 53 + 1700) / 1620;
	END_IF;
END_FUNCTION

FUNCTION DAY_OF_MONTH:INT
	VAR_INPUT
		IDATE :	UDINT;
	END_VAR

	day_of_month := DAY_OF_YEAR_UDINT(idate);

	IF leap_of_Date((idate)) THEN
		CASE day_of_month OF
			32..60	:	day_of_month := day_of_month - 31;
			61..91	:	day_of_month := day_of_month - 60;
			92..121 :	day_of_month := day_of_month - 91;
			122..152:	day_of_month := day_of_month - 121;
			153..182:	day_of_month := day_of_month - 152;
			183..213:	day_of_month := day_of_month - 182;
			214..244:	day_of_month := day_of_month - 213;
			245..274:	day_of_month := day_of_month - 244;
			275..305:	day_of_month := day_of_month - 274;
			306..335:	day_of_month := day_of_month - 305;
			336..366:	day_of_month := day_of_month - 335;
		END_CASE;
	ELSE
		CASE day_of_month OF
			32..59	:	day_of_month := day_of_month - 31;
			60..90	:	day_of_month := day_of_month - 59;
			91..120 :	day_of_month := day_of_month - 90;
			121..151:	day_of_month := day_of_month - 120;
			152..181:	day_of_month := day_of_month - 151;
			182..212:	day_of_month := day_of_month - 181;
			213..243:	day_of_month := day_of_month - 212;
			244..273:	day_of_month := day_of_month - 243;
			274..304:	day_of_month := day_of_month - 273;
			305..334:	day_of_month := day_of_month - 304;
			335..365:	day_of_month := day_of_month - 334;
		END_CASE;
	END_IF;
END_FUNCTION

FUNCTION DATE_ADD:UDINT
	VAR_INPUT
		IDATE :	UDINT;
		D :	INT;
		W :	INT;
		M :	INT;
		Y :	INT;
	END_VAR

	VAR
		mo :	INT;
		yr :	INT;
		dm :	INT;
	END_VAR

	DATE_ADD := IDATE + INT_TO_UDINT(D + W * 7) * UDINT#86400;
	yr := Y + YEAR_OF_DATE(DATE_ADD);
	mo := M + MONTH_OF_DATE(DATE_ADD);
	dm := DAY_OF_MONTH(DATE_ADD);
	WHILE mo > 12 DO
		mo := mo - 12;
		yr := yr + 1;
	END_WHILE;
	WHILE mo < 1 DO
		mo := mo + 12;
		yr := yr - 1;
	END_WHILE;
	DATE_ADD := SET_DATE(yr, mo, dm);
END_FUNCTION

FUNCTION DT_TO_DATE2:UDINT
	VAR_INPUT
		IN :	UDINT;
	END_VAR

	DT_TO_DATE2 := (IN / UDINT#86400) * UDINT#86400;
END_FUNCTION

FUNCTION DAY_OF_DATE:DINT
	VAR_INPUT
		IDATE :	UDINT;
	END_VAR

	day_of_date := UDINT_TO_DINT(idate / UDINT#86400);
END_FUNCTION

FUNCTION LEAP_YEAR:BOOL

  VAR_INPUT
    YEAR :	INT;
  END_VAR

  IF (year MOD INT#400) = INT#00 THEN
    leap_year := TRUE;
  ELSIF (year MOD INT#100) = INT#00 THEN
    leap_year := FALSE;
  ELSIF (year MOD INT#04) = INT#00 THEN
    leap_year := TRUE;
  ELSE
    leap_year := FALSE;
  END_IF;

END_FUNCTION

FUNCTION HOUR:INT
	VAR_INPUT
		ITOD :	UDINT;
	END_VAR
	hour := UDINT_TO_INT(itod / UDINT#3600000);
END_FUNCTION

FUNCTION SET_DT:UDINT

	VAR_INPUT
		YEAR : INT;
		MONTH :	INT;
		DAY : INT;
		HOURR : INT;
		MINUTE : INT;
		SECOND : INT;
	END_VAR

	SET_DT := SET_DATE(YEAR, MONTH, DAY) + _INT_TO_UDINT(SECOND) + _INT_TO_UDINT(MINUTE) * UDINT#60 + _INT_TO_UDINT(HOURR) * UDINT#3600;

END_FUNCTION

FUNCTION DST:BOOL
	VAR_INPUT
		UTC :	UDINT;
	END_VAR

	VAR
		yr :	INT;
		yr4 :	UDINT;
		ltc :	UDINT;
		idate :	UDINT;
	END_VAR

	yr := YEAR_OF_DATE(DT_TO_DATE2(UTC));
	ltc := UTC;
	idate := SET_DT(yr, 3, 31, 1, 0, 0);
	yr4 := DWORD_TO_UDINT(SHR(INT_TO_DWORD(5 * yr), 2)) + UDINT#1;
	DST := (idate - ((yr4 + UDINT#3) MOD UDINT#7) * UDINT#86400 <= ltc) AND (idate + (UDINT#214 - (yr4) MOD UDINT#7) * UDINT#86400 > ltc);

END_FUNCTION

FUNCTION UTC_TO_LTIME:UDINT

	VAR_INPUT
		UTC :	UDINT;
		DST_ENABLE :	BOOL;
		TIME_ZONE_OFFSET :	INT;
	END_VAR

	VAR
		tmp :	INT;
	END_VAR

	UTC_TO_LTIME := UTC + _INT_TO_UDINT(TIME_ZONE_OFFSET) * UDINT#60 + BOOL_TO_UDINT(DST_ENABLE AND DST(UTC)) * UDINT#3600;

	tmp := TIME_ZONE_OFFSET * 60 + BOOL_TO_INT(DST_ENABLE AND DST(UTC)) * 3600;
	IF tmp < 0 THEN
		UTC_TO_LTIME := UTC - _INT_TO_UDINT(ABS(tmp));
	ELSE
		UTC_TO_LTIME := UTC + _INT_TO_UDINT(tmp);
	END_IF;

END_FUNCTION

FUNCTION YEAR_BEGIN:UDINT
	VAR_INPUT
		Y :	INT;
	END_VAR
	year_begin := DWORD_TO_UDINT(SHR(UDINT_TO_DWORD(_INT_TO_UDINT(y) * UDINT#1461 - UDINT#2878169),2))*UDINT#86400;

END_FUNCTION

FUNCTION WORK_WEEK:INT

	VAR_INPUT
		IDATE :	UDINT;
	END_VAR

	VAR
		d1 :	UDINT;
		w1 :	INT;
		ds :	UDINT;
		yr :	INT;
		w31 :	INT;
		w01 :	INT;
		wm :	INT;
	END_VAR

	yr := YEAR_OF_DATE(idate);
	d1 := year_begin(yr);
	w1 := DAY_OF_WEEK(d1);
	IF w1 < 5 THEN
		ds := d1 - _INT_TO_UDINT(w1+6) * UDINT#86400;
	ELSE
		ds := d1 + _INT_TO_UDINT(1-w1) * UDINT#86400;
	END_IF;

	work_week := UDINT_TO_INT((idate - ds) / UDINT#604800);

	IF work_week = 0 THEN
		IF w1 > 1 THEN w31 := w1 - 1; ELSE W31 := 7; END_IF;
		IF leap_year(yr - 1) THEN IF w31 > 1 THEN w01 := W31 - 1; ELSE w1 := 7; END_IF; END_IF;
		WORK_WEEK := 52 + BOOL_TO_INT(w31 = 4 OR w01 = 4);
	ELSE
		IF leap_year(yr) THEN
			IF w1 < 7 THEN w31 := w1 + 1; ELSE w31 := 1; END_IF;
		ELSE
			w31 := w1;
		END_IF;
		wm := 52 + BOOL_TO_INT(w31 = 4 OR w1 = 4);
		IF work_week > wm THEN work_week := 1; END_IF;
	END_IF;

END_FUNCTION

FUNCTION_BLOCK HOLIDAY_Block
	VAR_INPUT
		DATE_IN :	UDINT;
		LANGU :	INT;
		FRIDAY :	BOOL;
		SATURDAY :	BOOL;
		SUNDAY :	BOOL;
	END_VAR

	VAR_IN_OUT
		HOLIDAYS :	oscat_HOLIDAY_DATA_0_29;
	END_VAR

	VAR_OUTPUT
		Y :	BOOL;
		NAME :	STRING;
	END_VAR

	VAR
		size :	INT := INT#29;
		last_active :	UDINT;
		ostern :	UDINT;
		i :	INT;
		jahr :	INT;
		x_date :	UDINT;
		lx :	INT;
		wdx :	INT;
		SETUP_LOCATIONS :	SETUP_LOCATION;
		SETUP_WEEKDAYSS :	SETUP_WEEKDAYS;
		SETUP_LANGUAGES :	SETUP_LANGUAGE_Block;
		LOCATION :	oscat_LOCATION;
		WEEKDAYS :	oscat_WEEKDAYS;
		LANGUAGE :	oscat_LANGUAGE;
		wd :	INT;
	END_VAR

	IF last_active = date_in THEN RETURN; END_IF;
	last_active := DATE_IN;

	SETUP_LOCATIONS(LOCATION:=LOCATION);
	LOCATION:=SETUP_LOCATIONS.LOCATION;

	SETUP_WEEKDAYSS(WEEKDAYS:=WEEKDAYS);
	WEEKDAYS:=SETUP_WEEKDAYSS.WEEKDAYS;

	SETUP_LANGUAGES(LANGUAGE:=LANGUAGE);
	LANGUAGE:=SETUP_LANGUAGES.LANGUAGE;

	IF LANGU = 0 THEN
		lx := language.DEFAULT;
	ELSE
		lx := MIN(language.LMAX, LANGU);
	END_IF;

	jahr := YEAR_OF_DATE(date_in);
	ostern := EASTER(jahr);
	wdx := DAY_OF_WEEK(DATE_IN);
	Y := FALSE;

	FOR i := 0 TO size DO
		x_date := SET_DATE(jahr, SINT_TO_INT(HOLIDAYS[i].MONTH) , SINT_TO_INT(HOLIDAYS[i].DAY));
		IF HOLIDAYS[i].USE = SINT#1 AND HOLIDAYS[i].MONTH > SINT#0 THEN
			(* check for fixed date holiday *)
			IF x_date = date_in THEN
				Y := TRUE;
				NAME := HOLIDAYS[i].NAME;
				RETURN;
			END_IF;
		ELSIF HOLIDAYS[i].USE = SINT#1 AND HOLIDAYS[i].MONTH = SINT#0 THEN
			(* check for holiday in reference to easter *)
			IF DATE_ADD(ostern, SINT_TO_INT(HOLIDAYS[i].DAY),0,0,0) = date_in THEN
				Y := TRUE;
				NAME := HOLIDAYS[i].NAME;
				RETURN;
			END_IF;
		ELSIF HOLIDAYS[i].USE < SINT#0 THEN
			(* check for holiday on a weekday before date *)
			IF DAY_OF_WEEK(date_in) = SINT_TO_INT(ABS(HOLIDAYS[i].USE)) AND date_in < x_date AND date_in >= DATE_ADD(x_date,-7,0,0,0) THEN
				Y := TRUE;
				NAME := HOLIDAYS[i].NAME;
				RETURN;
			END_IF;
		END_IF;
	END_FOR;

	IF NOT Y AND (wdx = 5 AND FRIDAY OR wdx = 6 AND SATURDAY OR wdx = 7 AND SUNDAY) THEN
		Y := TRUE;
		wd := LOCATION.LANGUAGE[lx];
		NAME := WEEKDAYS[wd][wdx];
	ELSE
		NAME := '';
	END_IF;
END_FUNCTION_BLOCK

FUNCTION_BLOCK CALENDAR_CALC
	VAR_INPUT
		SPE :	BOOL;
		H :	REAL := REAL#-0.83333333333;
	END_VAR

	VAR_IN_OUT
		XCAL :	oscat_CALENDAR;
		HOLIDAYS :	oscat_HOLIDAY_DATA_0_29;
	END_VAR

	VAR
		last :	UDINT;
		last_day :	DINT;
		holy :	HOLIDAY_Block;
		sun :	SUN_TIME_Block;
		last_hour :	INT;
		utod :	UDINT;
		pos :	SUN_POS;
		plast :	UDINT;
		dtemp :	DINT;
		tmp :	INT;
		SETUP_LOCATIONS :	SETUP_LOCATION;
		LOCATION :	oscat_LOCATION;
	END_VAR

	IF xcal.UTC <> last THEN
		last := XCAL.UTC;
		utod := DT_TO_TOD2(xcal.UTC);

		XCAL.LDT := UTC_TO_LTIME(XCAL.UTC, XCAL.DST_EN, XCAL.OFFSET);
		XCAL.LDATE := DT_TO_DATE2(XCAL.LDT);
		XCAL.LTOD := DT_TO_TOD2(XCAL.LDT);
		dtemp := DAY_OF_DATE(XCAL.LDATE);
		xcal.night := XCAL.LTOD < XCAL.SUN_RISE OR XCAL.LTOD > XCAL.SUN_SET;

		tmp := HOUR(xcal.LTOD);
		IF  tmp <> last_hour THEN
			XCAL.DST_ON := DST(XCAL.UTC) AND xcal.DST_EN;
			last_hour := tmp;
		END_IF;

		IF dtemp <> last_day THEN
			SETUP_LOCATIONS(LOCATION:=LOCATION);
			LOCATION:=SETUP_LOCATIONS.LOCATION;

			last_day := dtemp;
			XCAL.YEAR := YEAR_OF_DATE(XCAL.LDATE);
			XCAL.MONTH := MONTH_OF_DATE(XCAL.LDATE);
			XCAL.DAY := DAY_OF_MONTH(XCAL.LDATE);
			XCAL.WEEKDAY := DAY_OF_WEEK(XCAL.LDATE);
			HOLY(date_in := XCAL.LDATE, LANGU := xcal.LANGUAGE, HOLIDAYS := HOLIDAYS);
			HOLIDAYS := HOLY.HOLIDAYS;
			XCAL.HOLIDAY := HOLY.Y;
			XCAL.HOLY_NAME := HOLY.NAME;
			sun(latitude := XCAL.LATITUDE, longitude := xcal.LONGITUDE, utc := DT_TO_DATE2(xcal.UTC), H := H);
			XCAL.SUN_RISE := DINT_TO_UDINT(UDINT_TO_DINT(sun.sun_rise) + INT_TO_DINT(XCAL.OFFSET) * DINT#60000 + SEL_DINT(XCAL.DST_ON,DINT#0,DINT#3600000));
			XCAL.SUN_SET := DINT_TO_UDINT(UDINT_TO_DINT(sun.sun_set) + INT_TO_DINT(XCAL.OFFSET) * DINT#60000 + SEL_DINT(XCAL.DST_ON,DINT#0,DINT#3600000));
			XCAL.SUN_MIDDAY := DINT_TO_UDINT(UDINT_TO_DINT(sun.midday) + INT_TO_DINT(XCAL.OFFSET) * DINT#60000 + SEL_DINT(XCAL.DST_ON,DINT#0,DINT#3600000));
			XCAL.SUN_HEIGTH := sun.sun_declination;
			XCAL.WORK_WEEK := WORK_WEEK(XCAL.LDATE);
		END_IF;

		IF SPE AND xcal.UTC -  plast >= TIME_TO_UDINT2(t#25s) THEN
			plast := last;
			pos(latitude := xcal.LATITUDE, longitude := xcal.LONGITUDE, utc := xcal.UTC);
			xcal.SUN_HOR := pos.B;
			xcal.SUN_VER := pos.HR;
		END_IF;
	END_IF;
END_FUNCTION_BLOCK

PROGRAM program0
  VAR
    LocalVar0 : BOOL;
    LocalVar1 : REAL;
	LocalVar2 : oscat_CALENDAR;
	LocalVar3 : oscat_HOLIDAY_DATA_0_29;
	func_block : CALENDAR_CALC;
  END_VAR
	func_block.SPE  := LocalVar0;
	func_block.H := LocalVar1;
	func_block.XCAL  := LocalVar2;
	func_block.HOLIDAYS := LocalVar3;
	func_block();
	LocalVar2 := func_block.XCAL;
	LocalVar3 := func_block.HOLIDAYS;

END_PROGRAM

CONFIGURATION Config0
	RESOURCE Res0 ON PLC
		TASK task0(INTERVAL := T#20ms,PRIORITY := 0);
		PROGRAM instance0 WITH task0 : program0;
	END_RESOURCE
END_CONFIGURATION

(* ---- CALIBRATE.ST ---- *)
FUNCTION_BLOCK CALIBRATE
	VAR_INPUT
		X :	REAL;
		CO :	BOOL;
		CS :	BOOL;
		Y_OFFSET :	REAL;
		Y_SCALE :	REAL;
	END_VAR

	VAR_OUTPUT
		Y :	REAL;
	END_VAR

	VAR RETAIN
		offset :	REAL;
		Scale :	REAL := 1.0;
	END_VAR

	IF CO THEN
		OFFSET := Y_Offset - X;
	ELSIF CS THEN
		SCALE := Y_scale / (X + OFFSET);
	END_IF;
	Y := (X + OFFSET) * SCALE;

END_FUNCTION_BLOCK

PROGRAM program0
  VAR
    LocalVar0 : REAL;
    LocalVar1 : BOOL;
	LocalVar2 : BOOL;
	LocalVar3 : REAL;
	LocalVar4 : REAL;
	LocalOUT  : REAL;
	func_block : CALIBRATE;
  END_VAR
	func_block.X  := LocalVar0;
	func_block.CO := LocalVar1;
	func_block.CS  := LocalVar2;
	func_block.Y_OFFSET := LocalVar3;
	func_block.Y_SCALE := LocalVar4;
	func_block();
	LocalOUT := func_block.Y;

END_PROGRAM

CONFIGURATION Config0
  RESOURCE Res0 ON PLC
    TASK task0(INTERVAL := T#20ms,PRIORITY := 0);
    PROGRAM instance0 WITH task0 : program0;
  END_RESOURCE
END_CONFIGURATION

(* ---- CARG.ST ---- *)
TYPE oscat_complex :
  STRUCT
	re : REAL;
	im : REAL;
  END_STRUCT;
END_TYPE

FUNCTION ATAN2:REAL
	VAR_INPUT
		X :	REAL;
		Y :	REAL;
	END_VAR

	IF X > 0.0 THEN
		ATAN2 := ATAN(Y/X);
	ELSIF X < 0.0 THEN
		IF Y >= 0.0 THEN
			ATAN2 := ATAN(Y/X) + 3.14159265358979323846264338327950288;
		ELSE
			ATAN2 := ATAN(Y/X) - 3.14159265358979323846264338327950288;
		END_IF;
	ELSIF Y > 0.0 THEN
		ATAN2 := 1.5707963267948965580;
	ELSIF Y < 0.0 THEN
		ATAN2 := -1.5707963267948965580;
	ELSE
		ATAN2 := 0.0;
	END_IF;

END_FUNCTION

FUNCTION_BLOCK CARG_Block

	VAR_INPUT
		X :	oscat_complex;
	END_VAR

	VAR_OUTPUT
		CARG :	REAL;
	END_VAR

	CARG := ATAN2(X.im, X.re);

END_FUNCTION_BLOCK

PROGRAM program0
  VAR
    LocalVar0 : oscat_complex;
	LocalOUT  : REAL;
	func_block : CARG_Block;
  END_VAR
	func_block.X  := LocalVar0;
	func_block();
	LocalOUT := func_block.CARG;
END_PROGRAM

CONFIGURATION Config0
  RESOURCE Res0 ON PLC
    TASK task0(INTERVAL := T#20ms,PRIORITY := 0);
    PROGRAM instance0 WITH task0 : program0;
  END_RESOURCE
END_CONFIGURATION

(* ---- CASIN.ST ---- *)
TYPE oscat_complex :
  STRUCT
	re : REAL;
	im : REAL;
  END_STRUCT;
END_TYPE

FUNCTION ATAN2:REAL
	VAR_INPUT
		X :	REAL;
		Y :	REAL;
	END_VAR

	IF X > 0.0 THEN
		ATAN2 := ATAN(Y/X);
	ELSIF X < 0.0 THEN
		IF Y >= 0.0 THEN
			ATAN2 := ATAN(Y/X) + 3.14159265358979323846264338327950288;
		ELSE
			ATAN2 := ATAN(Y/X) - 3.14159265358979323846264338327950288;
		END_IF;
	ELSIF Y > 0.0 THEN
		ATAN2 := 1.5707963267948965580;
	ELSIF Y < 0.0 THEN
		ATAN2 := -1.5707963267948965580;
	ELSE
		ATAN2 := 0.0;
	END_IF;

END_FUNCTION

FUNCTION HYPOT:REAL
	VAR_INPUT
		X :	REAL;
		Y :	REAL;
	END_VAR

	HYPOT := SQRT(x*x + y*y);
END_FUNCTION

FUNCTION_BLOCK CLOG_Block

	VAR_INPUT
		X :	oscat_complex;
	END_VAR

	VAR_OUTPUT
		CLOG :	oscat_complex;
	END_VAR

	CLOG.re := LN(HYPOT(X.re, X.im));
	CLOG.im := ATAN2(X.im, X.re);

END_FUNCTION_BLOCK

FUNCTION SGN : INT
  VAR_INPUT
    x : REAL;
  END_VAR

  IF X > 0.0 THEN
  	sgn := 1;
  ELSIF X < 0.0 THEN
  	sgn := -1;
  ELSE
  	sgn := 0;
  END_IF;
END_FUNCTION

FUNCTION_BLOCK CSQRT_Block
	VAR_INPUT
		X :	oscat_complex;
	END_VAR

	VAR_OUTPUT
		CSQRT :	oscat_complex;
	END_VAR

	VAR
		temp :	REAL;
	END_VAR

	temp := HYPOT(x.re, x.im);
	CSQRT.re :=  SQRT(0.5 * (temp + x.re));
	CSQRT.im :=  INT_TO_REAL(sgn(x.im)) * SQRT(0.5 * (temp - x.re));

END_FUNCTION_BLOCK

FUNCTION_BLOCK CASINH_Block
	VAR_INPUT
		X :	oscat_complex;
	END_VAR

	VAR_OUTPUT
		CASINH :	oscat_complex;
	END_VAR

	VAR
		Y :	oscat_complex;
		CLOG :	CLOG_Block;
		CSQRT :	CSQRT_Block;
	END_VAR

	y.re := (X.re - X.im)*(X.re + X.im) + 1.0;
	y.im := 2.0 * X.re * X.im;
	CSQRT(X:=y);
	y    := CSQRT.CSQRT;
	y.re := y.re + x.re;
	y.im := y.im + x.im;
	CLOG(X:=y);
	CASINH  := CLOG.CLOG;
END_FUNCTION_BLOCK

FUNCTION_BLOCK CASIN_Block
	VAR_INPUT
		X :	oscat_complex;
	END_VAR

	VAR_OUTPUT
		CASIN :	oscat_complex;
	END_VAR

	VAR
		Y :	oscat_complex;
		CASINH :	CASINH_Block;
	END_VAR

	y.re := -x.im;
	y.im := x.re;
	CASINH(X:=y);
	y := CASINH.CASINH;
	CASIN.re := y.im;
	CASIN.im := -y.re;
END_FUNCTION_BLOCK

PROGRAM program0
  VAR
    LocalVar0 : oscat_complex;
	LocalOUT  : oscat_complex;
	func_block : CASIN_Block;
  END_VAR
	func_block.X  := LocalVar0;
	func_block();
	LocalOUT := func_block.CASIN;
END_PROGRAM

CONFIGURATION Config0
  RESOURCE Res0 ON PLC
    TASK task0(INTERVAL := T#20ms,PRIORITY := 0);
    PROGRAM instance0 WITH task0 : program0;
  END_RESOURCE
END_CONFIGURATION

(* ---- CASINH.ST ---- *)
TYPE oscat_complex :
  STRUCT
	re : REAL;
	im : REAL;
  END_STRUCT;
END_TYPE

FUNCTION ATAN2:REAL
	VAR_INPUT
		X :	REAL;
		Y :	REAL;
	END_VAR

	IF X > 0.0 THEN
		ATAN2 := ATAN(Y/X);
	ELSIF X < 0.0 THEN
		IF Y >= 0.0 THEN
			ATAN2 := ATAN(Y/X) + 3.14159265358979323846264338327950288;
		ELSE
			ATAN2 := ATAN(Y/X) - 3.14159265358979323846264338327950288;
		END_IF;
	ELSIF Y > 0.0 THEN
		ATAN2 := 1.5707963267948965580;
	ELSIF Y < 0.0 THEN
		ATAN2 := -1.5707963267948965580;
	ELSE
		ATAN2 := 0.0;
	END_IF;

END_FUNCTION

FUNCTION HYPOT:REAL
	VAR_INPUT
		X :	REAL;
		Y :	REAL;
	END_VAR

	HYPOT := SQRT(x*x + y*y);
END_FUNCTION

FUNCTION_BLOCK CLOG_Block

	VAR_INPUT
		X :	oscat_complex;
	END_VAR

	VAR_OUTPUT
		CLOG :	oscat_complex;
	END_VAR

	CLOG.re := LN(HYPOT(X.re, X.im));
	CLOG.im := ATAN2(X.im, X.re);

END_FUNCTION_BLOCK

FUNCTION SGN : INT
  VAR_INPUT
    x : REAL;
  END_VAR

  IF X > 0.0 THEN
  	sgn := 1;
  ELSIF X < 0.0 THEN
  	sgn := -1;
  ELSE
  	sgn := 0;
  END_IF;
END_FUNCTION

FUNCTION_BLOCK CSQRT_Block
	VAR_INPUT
		X :	oscat_complex;
	END_VAR

	VAR_OUTPUT
		CSQRT :	oscat_complex;
	END_VAR

	VAR
		temp :	REAL;
	END_VAR

	temp := HYPOT(x.re, x.im);
	CSQRT.re :=  SQRT(0.5 * (temp + x.re));
	CSQRT.im :=  INT_TO_REAL(sgn(x.im)) * SQRT(0.5 * (temp - x.re));

END_FUNCTION_BLOCK

FUNCTION_BLOCK CASINH_Block
	VAR_INPUT
		X :	oscat_complex;
	END_VAR

	VAR_OUTPUT
		CASINH :	oscat_complex;
	END_VAR

	VAR
		Y :	oscat_complex;
		CLOG :	CLOG_Block;
		CSQRT :	CSQRT_Block;
	END_VAR

	y.re := (X.re - X.im)*(X.re + X.im) + 1.0;
	y.im := 2.0 * X.re * X.im;
	CSQRT(X:=y);
	y    := CSQRT.CSQRT;
	y.re := y.re + x.re;
	y.im := y.im + x.im;
	CLOG(X:=y);
	CASINH  := CLOG.CLOG;
END_FUNCTION_BLOCK

PROGRAM program0
  VAR
    LocalVar0 : oscat_complex;
	LocalOUT  : oscat_complex;
	func_block : CASINH_Block;
  END_VAR
	func_block.X  := LocalVar0;
	func_block();
	LocalOUT := func_block.CASINH;
END_PROGRAM

CONFIGURATION Config0
  RESOURCE Res0 ON PLC
    TASK task0(INTERVAL := T#20ms,PRIORITY := 0);
    PROGRAM instance0 WITH task0 : program0;
  END_RESOURCE
END_CONFIGURATION

(* ---- CATAN.ST ---- *)
TYPE oscat_complex :
  STRUCT
	re : REAL;
	im : REAL;
  END_STRUCT;
END_TYPE

FUNCTION_BLOCK CATAN_Block
	VAR_INPUT
		X :	oscat_complex;
	END_VAR

	VAR_OUTPUT
		CATAN :	oscat_complex;
	END_VAR

	VAR
		r2 :	REAL;
		num :	REAL;
		den :	REAL;
	END_VAR

	r2 := x.re * x.re;
	den := 1.0 - r2 - x.im * x.im;
	CATAN.re := 0.5 * ATAN(2.0 * x.re / den);
	num := x.im + 1.0;
	num := r2 + num * num;
	den := x.im - 1.0;
	den := r2 + den * den;
	CATAN.im := 0.25 * (LN(num)-LN(den));

END_FUNCTION_BLOCK

PROGRAM program0
  VAR
    LocalVar0 : oscat_complex;
	LocalOUT  : oscat_complex;
	func_block : CATAN_Block;
  END_VAR
	func_block.X  := LocalVar0;
	func_block();
	LocalOUT := func_block.CATAN;
END_PROGRAM

CONFIGURATION Config0
  RESOURCE Res0 ON PLC
    TASK task0(INTERVAL := T#20ms,PRIORITY := 0);
    PROGRAM instance0 WITH task0 : program0;
  END_RESOURCE
END_CONFIGURATION

(* ---- CATANH.ST ---- *)
TYPE oscat_complex :
  STRUCT
	re : REAL;
	im : REAL;
  END_STRUCT;
END_TYPE

FUNCTION_BLOCK CATANH_Block
	VAR_INPUT
		X :	oscat_complex;
	END_VAR

	VAR_OUTPUT
		CATANH :	oscat_complex;
	END_VAR

	VAR
		i2 :	REAL;
		num :	REAL;
		den :	REAL;
	END_VAR

	i2 := x.im * x.im;
	num := 1.0 + x.re;
	num := i2 + num * num;
	den := 1.0 - x.re;
	den := i2 + den * den;
	CATANH.re := 0.25 * (LN(num) - LN(den));
	den := 1.0 - x.re * x.re - i2;
	CATANH.im := 0.5 * ATAN(2.0 * x.im / den);

END_FUNCTION_BLOCK

PROGRAM program0
  VAR
    LocalVar0 : oscat_complex;
	LocalOUT  : oscat_complex;
	func_block : CATANH_Block;
  END_VAR
	func_block.X  := LocalVar0;
	func_block();
	LocalOUT := func_block.CATANH;
END_PROGRAM

CONFIGURATION Config0
  RESOURCE Res0 ON PLC
    TASK task0(INTERVAL := T#20ms,PRIORITY := 0);
    PROGRAM instance0 WITH task0 : program0;
  END_RESOURCE
END_CONFIGURATION

(* ---- CCON.ST ---- *)
TYPE oscat_complex :
  STRUCT
	re : REAL;
	im : REAL;
  END_STRUCT;
END_TYPE

FUNCTION_BLOCK CCON_Block

	VAR_INPUT
		X :	oscat_complex;
	END_VAR

	VAR_OUTPUT
		CCON :	oscat_complex;
	END_VAR

	CCON.re := x.re;
	CCON.im := -x.im;

END_FUNCTION_BLOCK

PROGRAM program0
  VAR
    LocalVar0 : oscat_complex;
	LocalOUT  : oscat_complex;
	func_block : CCON_Block;
  END_VAR
	func_block.X  := LocalVar0;
	func_block();
	LocalOUT := func_block.CCON;
END_PROGRAM

CONFIGURATION Config0
  RESOURCE Res0 ON PLC
    TASK task0(INTERVAL := T#20ms,PRIORITY := 0);
    PROGRAM instance0 WITH task0 : program0;
  END_RESOURCE
END_CONFIGURATION

(* ---- CCOS.ST ---- *)
TYPE oscat_complex :
  STRUCT
	re : REAL;
	im : REAL;
  END_STRUCT;
END_TYPE

FUNCTION COSH:REAL
	VAR_INPUT
		X :	REAL;
	END_VAR

	VAR
		t :	REAL;
	END_VAR

	T := EXP(X);
	COSH := (1.0 / T + T) * 0.5;
END_FUNCTION

FUNCTION SINH:REAL
	VAR_INPUT
		X :	REAL;
	END_VAR

	IF ABS(x) < 2.0E-3 THEN
		SINH := X;
	ELSE
		SINH := (EXP(x) - EXP(-x)) * 0.5;
	END_IF;
END_FUNCTION

FUNCTION_BLOCK CCOSH_Block
	VAR_INPUT
		X :	oscat_complex;
	END_VAR

	VAR_OUTPUT
		CCOSH :	oscat_complex;
	END_VAR

	CCOSH.re := cosH(x.re) * COS(x.im);
	CCOSH.im := sinH(x.re) * SIN(x.im);
END_FUNCTION_BLOCK

FUNCTION_BLOCK CSET_Block
	VAR_INPUT
		RE :	REAL;
		IM :	REAL;
	END_VAR

	VAR_OUTPUT
		CSET :	oscat_complex;
	END_VAR

	CSET.re := RE;
	CSET.im := IM;
END_FUNCTION_BLOCK

FUNCTION_BLOCK CCOS_Block
	VAR_INPUT
		X :	oscat_complex;
	END_VAR

	VAR_OUTPUT
		CCOS :	oscat_complex;
	END_VAR

	VAR
		CSET :	CSET_Block;
		CCOSH :	CCOSH_Block;
	END_VAR

	CSET(RE:= -X.im,IM:=X.re);
	CCOSH(X:=CSET.CSET);
	CCOS := CCOSH.CCOSH;

END_FUNCTION_BLOCK

PROGRAM program0
  VAR
    LocalVar0 : oscat_complex;
	LocalOUT  : oscat_complex;
	func_block : CCOS_Block;
  END_VAR
	func_block.X  := LocalVar0;
	func_block();
	LocalOUT := func_block.CCOS;
END_PROGRAM

CONFIGURATION Config0
  RESOURCE Res0 ON PLC
    TASK task0(INTERVAL := T#20ms,PRIORITY := 0);
    PROGRAM instance0 WITH task0 : program0;
  END_RESOURCE
END_CONFIGURATION

(* ---- CCOSH.ST ---- *)
TYPE oscat_complex :
  STRUCT
	re : REAL;
	im : REAL;
  END_STRUCT;
END_TYPE

FUNCTION COSH:REAL
	VAR_INPUT
		X :	REAL;
	END_VAR

	VAR
		t :	REAL;
	END_VAR

	T := EXP(X);
	COSH := (1.0 / T + T) * 0.5;
END_FUNCTION

FUNCTION SINH:REAL
	VAR_INPUT
		X :	REAL;
	END_VAR

	IF ABS(x) < 2.0E-3 THEN
		SINH := X;
	ELSE
		SINH := (EXP(x) - EXP(-x)) * 0.5;
	END_IF;
END_FUNCTION

FUNCTION_BLOCK CCOSH_Block
	VAR_INPUT
		X :	oscat_complex;
	END_VAR

	VAR_OUTPUT
		CCOSH :	oscat_complex;
	END_VAR

	CCOSH.re := cosH(x.re) * COS(x.im);
	CCOSH.im := sinH(x.re) * SIN(x.im);
END_FUNCTION_BLOCK

PROGRAM program0
  VAR
    LocalVar0 : oscat_complex;
	LocalOUT  : oscat_complex;
	func_block : CCOSH_Block;
  END_VAR
	func_block.X  := LocalVar0;
	func_block();
	LocalOUT := func_block.CCOSH;
END_PROGRAM

CONFIGURATION Config0
  RESOURCE Res0 ON PLC
    TASK task0(INTERVAL := T#20ms,PRIORITY := 0);
    PROGRAM instance0 WITH task0 : program0;
  END_RESOURCE
END_CONFIGURATION

(* ---- CDIV.ST ---- *)
TYPE oscat_complex :
  STRUCT
	re : REAL;
	im : REAL;
  END_STRUCT;
END_TYPE

FUNCTION_BLOCK CDIV_Block

	VAR_INPUT
		X :	oscat_complex;
		Y :	oscat_complex;
	END_VAR

	VAR_OUTPUT
		CDIV :	oscat_complex;
	END_VAR

	VAR
		temp :	REAL;
	END_VAR

	temp := Y.re * Y.re + Y.im * Y.im;
	IF temp = 0.0 THEN CDIV.re := 0.0;CDIV.im := 0.0;RETURN;END_IF;
	CDIV.re := (X.re * Y.re + X.im * Y.im) / temp;
	CDIV.im := (X.im * Y.re - X.re * Y.im) / temp;

END_FUNCTION_BLOCK

PROGRAM program0

	VAR
		X :	oscat_complex;
		Y :	oscat_complex;

		CDIV :	oscat_complex;

		func_block : CDIV_Block;
	END_VAR
	func_block.X := X;
	func_block.Y := Y;
	func_block();
	CDIV := func_block.CDIV;

END_PROGRAM

CONFIGURATION Config0

	RESOURCE Res0 ON PLC
		TASK task0(INTERVAL := T#20ms,PRIORITY := 0);
		PROGRAM instance0 WITH task0 : program0;
	END_RESOURCE

END_CONFIGURATION
